# B&R Automation Studio project Parker_BMM_ST_V5_3147_V12 (part 21)

```c
					/*-------------F5---------*/
					//					gPanelObj.idxKeyPicture[S$KEYMATRIX_F5] = STATE_INACTIVE;
					gPanelObj.idxKeyPicture[S$KEYMATRIX_F5] = STATE_SUB_PAGE;
					if(1 == EDGEPOS(gPanelObj.KeyMatric[S$KEYMATRIX_F5],KeyMatric[S$KEYMATRIX_F5]))
					{
					gPanelObj.SetPicture = PIC_BLOW_PIN_CONFIG;
				}
				if(gPanelObj.GetPicture == PIC_BLOW_PIN_CONFIG)gPanelObj.idxKeyPicture[S$KEYMATRIX_F5] = STATE_ACTIVE;

					/*------------F6-----------*/
					gPanelObj.idxKeyPicture[S$KEYMATRIX_F6] = STATE_SUB_PAGE;
					if(1 == EDGEPOS(gPanelObj.KeyMatric[S$KEYMATRIX_F6],KeyMatric[S$KEYMATRIX_F6]))
					{
					gPanelObj.SetPicture = PIC_EXTRLIFT_CONFIG;
				}
				if(gPanelObj.GetPicture == PIC_EXTRLIFT_CONFIG)gPanelObj.idxKeyPicture[S$KEYMATRIX_F6] = STATE_ACTIVE;

					/*------------F7-----------*/
					gPanelObj.idxKeyPicture[S$KEYMATRIX_F7] = STATE_INACTIVE;

					/*-----------F8------------*/
					gPanelObj.idxKeyPicture[S$KEYMATRIX_F8] = STATE_INACTIVE;

					/*----------F9-------------*/
					gPanelObj.idxKeyPicture[S$KEYMATRIX_F9] = STATE_INACTIVE;

					/*----------F10-------------*/
					gPanelObj.idxKeyPicture[S$KEYMATRIX_F10] = STATE_INACTIVE;

					/*----------F11-------------*/
					gPanelObj.idxKeyPicture[S$KEYMATRIX_F11] = STATE_SUB_PAGE;
					if(1 == EDGEPOS(gPanelObj.KeyMatric[S$KEYMATRIX_F11],KeyMatric[S$KEYMATRIX_F11]))
					{
					gPanelObj.SetPicture = PIC_CLAMP_TOGGLE;
				}
				if(gPanelObj.GetPicture == PIC_CLAMP_TOGGLE)gPanelObj.idxKeyPicture[S$KEYMATRIX_F11] = STATE_ACTIVE;

					/*----------F12-------------*/
					gPanelObj.idxKeyPicture[S$KEYMATRIX_F12] = STATE_SUB_PAGE;
					if(1 == EDGEPOS(gPanelObj.KeyMatric[S$KEYMATRIX_F12],KeyMatric[S$KEYMATRIX_F12]))
					{
					gPanelObj.SetPicture = PIC_CARRIAGE_TOGGLE;
				}
				if(gPanelObj.GetPicture == PIC_CARRIAGE_TOGGLE)gPanelObj.idxKeyPicture[S$KEYMATRIX_F12] = STATE_ACTIVE;

					/*----------F13-------------*/
					gPanelObj.idxKeyPicture[S$KEYMATRIX_F13] = STATE_SUB_PAGE;
					if(1 == EDGEPOS(gPanelObj.KeyMatric[S$KEYMATRIX_F13],KeyMatric[S$KEYMATRIX_F13]))
					{
					gPanelObj.SetPicture = PIC_EXTRLIFT_TOGGLE;
				}
				if(gPanelObj.GetPicture == PIC_EXTRLIFT_TOGGLE)gPanelObj.idxKeyPicture[S$KEYMATRIX_F13] = STATE_ACTIVE;

					/*----------F14-------------*/
					gPanelObj.idxKeyPicture[S$KEYMATRIX_F14] = STATE_SUB_PAGE;
					if(1 == EDGEPOS(gPanelObj.KeyMatric[S$KEYMATRIX_F14],KeyMatric[S$KEYMATRIX_F14]))
					{
					gPanelObj.SetPicture = PIC_CONFIG_HELP;
				}
				if(gPanelObj.GetPicture == PIC_CONFIG_HELP)gPanelObj.idxKeyPicture[S$KEYMATRIX_F14] = STATE_ACTIVE;

					/*----------F15-------------*/
					gPanelObj.idxKeyPicture[S$KEYMATRIX_F15] = STATE_SUB_PAGE;
					if(1 == EDGEPOS(gPanelObj.KeyMatric[S$KEYMATRIX_F15],KeyMatric[S$KEYMATRIX_F15]))
					{
					gPanelObj.SetPicture = PIC_CLAMP_L;
					if(1 == bHideLeftStation)gPanelObj.SetPicture = PIC_CLAMP_R;
				}

				/*----------F16-------------*/
				gPanelObj.idxKeyPicture[S$KEYMATRIX_F16] = STATE_SUB_PAGE;
					if(1 == EDGEPOS(gPanelObj.KeyMatric[S$KEYMATRIX_F16],KeyMatric[S$KEYMATRIX_F16]))
					{
					gPanelObj.SetPicture = PIC_PASSWORD_LOGIN;
				}

				break;

			case PIC_RECIPE:
				if(ChangePageDly > 0)
				{
					ChangePageDly--;
					break;
				}

				gPanelObj.idxKeyPicture[S$KEYMATRIX_F1] = STATE_SUB_PAGE;
					if(1 == EDGEPOS(gPanelObj.KeyMatric[S$KEYMATRIX_F1],KeyMatric[S$KEYMATRIX_F1]))
					{
					gPanelObj.SetPicture = PIC_OVERVIEW;
				}

				gPanelObj.idxKeyPicture[S$KEYMATRIX_F2] = STATE_SUB_PAGE;
					if(1 == EDGEPOS(gPanelObj.KeyMatric[S$KEYMATRIX_F2],KeyMatric[S$KEYMATRIX_F2]))
					{
					gPanelObj.SetPicture = gPanelObj.OldPicture;
				}

				gPanelObj.idxKeyPicture[S$KEYMATRIX_F3] = STATE_INACTIVE;

					if(1 == gRecipeOperate.usbDiskOk)
				{
					gPanelObj.idxKeyPicture[S$KEYMATRIX_F4] = STATE_SUB_BUTTON;
						gPanelObj.idxKeyPicture[S$KEYMATRIX_F5] = STATE_SUB_BUTTON;
						}
				else
				{
					gPanelObj.idxKeyPicture[S$KEYMATRIX_F4] = STATE_INACTIVE;
						gPanelObj.idxKeyPicture[S$KEYMATRIX_F5] = STATE_INACTIVE;
						}
				gPanelObj.idxKeyPicture[S$KEYMATRIX_F6] = STATE_INACTIVE;

					gPanelObj.idxKeyPicture[S$KEYMATRIX_F7] = STATE_INACTIVE;
					gPanelObj.idxKeyPicture[S$KEYMATRIX_F8] = STATE_INACTIVE;
					gPanelObj.idxKeyPicture[S$KEYMATRIX_F9] = STATE_INACTIVE;
					gPanelObj.idxKeyPicture[S$KEYMATRIX_F10] = STATE_INACTIVE;
					gPanelObj.idxKeyPicture[S$KEYMATRIX_F11] = STATE_SUB_BUTTON;
					gPanelObj.idxKeyPicture[S$KEYMATRIX_F12] = STATE_SUB_BUTTON;
					gPanelObj.idxKeyPicture[S$KEYMATRIX_F13] = STATE_SUB_BUTTON;
					gPanelObj.idxKeyPicture[S$KEYMATRIX_F14] = STATE_SUB_BUTTON;

					gPanelObj.idxKeyPicture[S$KEYMATRIX_F15] = STATE_INACTIVE;

					gPanelObj.idxKeyPicture[S$KEYMATRIX_F16] = STATE_SUB_PAGE;
					if(1 == EDGEPOS(gPanelObj.KeyMatric[S$KEYMATRIX_F16],KeyMatric[S$KEYMATRIX_F16]))
					{
					gPanelObj.SetPicture = PIC_PASSWORD_LOGIN;
				}
				break;

			//				case PIC_SPEED:
			//					if(ChangePageDly > 0)
			//					{
			//						ChangePageDly--;
			//						break;
			//					}
			//
			//					gPanelObj.idxKeyPicture[S$KEYMATRIX_F1] = STATE_SUB_PAGE;
			//						if(1 == EDGEPOS(gPanelObj.KeyMatric[S$KEYMATRIX_F1],KeyMatric[S$KEYMATRIX_F1]))
			//						{
			//						gPanelObj.SetPicture = PIC_OVERVIEW;
			//					}
			//
			//					gPanelObj.idxKeyPicture[S$KEYMATRIX_F2] = STATE_SUB_PAGE;
			//						if(1 == EDGEPOS(gPanelObj.KeyMatric[S$KEYMATRIX_F2],KeyMatric[S$KEYMATRIX_F2]))
			//						{
			//						gPanelObj.SetPicture = gPanelObj.OldPicture;
			//					}
			//
			//					gPanelObj.idxKeyPicture[S$KEYMATRIX_F3] = STATE_INACTIVE;
			////						if(1 == EDGEPOS(gPanelObj.KeyMatric[S$KEYMATRIX_F3],KeyMatric[S$KEYMATRIX_F3]))
			////						{
			////						gPanelObj.SetPicture =PIC_LENGTH;
			////					}
			//
			//					gPanelObj.idxKeyPicture[S$KEYMATRIX_F4] = STATE_INACTIVE;
			//						gPanelObj.idxKeyPicture[S$KEYMATRIX_F5] = STATE_INACTIVE;
			//						gPanelObj.idxKeyPicture[S$KEYMATRIX_F6] = STATE_INACTIVE;
			//						gPanelObj.idxKeyPicture[S$KEYMATRIX_F7] = STATE_INACTIVE;
			//						gPanelObj.idxKeyPicture[S$KEYMATRIX_F8] = STATE_INACTIVE;
			//
			//						gPanelObj.idxKeyPicture[S$KEYMATRIX_F9] = STATE_SUB_PAGE;
			//						if(1 == EDGEPOS(gPanelObj.KeyMatric[S$KEYMATRIX_F9],KeyMatric[S$KEYMATRIX_F9]))
			//						{
			//						gPanelObj.SetPicture = PIC_TEMP_CONSTRUCT;
			//					}
			//
			//					gPanelObj.idxKeyPicture[S$KEYMATRIX_F10] = STATE_SUB_PAGE;
			//						if(1 == EDGEPOS(gPanelObj.KeyMatric[S$KEYMATRIX_F10],KeyMatric[S$KEYMATRIX_F10]))
			//						{
			//						gPanelObj.SetPicture =PIC_THICK_START;
			//					}
			//
			//					gPanelObj.idxKeyPicture[S$KEYMATRIX_F11] = STATE_INACTIVE;
			//						gPanelObj.idxKeyPicture[S$KEYMATRIX_F12] = STATE_INACTIVE;
			//						gPanelObj.idxKeyPicture[S$KEYMATRIX_F13] = STATE_INACTIVE;
			//						gPanelObj.idxKeyPicture[S$KEYMATRIX_F14] = STATE_INACTIVE;
			//						gPanelObj.idxKeyPicture[S$KEYMATRIX_F15] = STATE_INACTIVE;
			//
			//						gPanelObj.idxKeyPicture[S$KEYMATRIX_F16] = STATE_SUB_PAGE;
			//						if(1 == EDGEPOS(gPanelObj.KeyMatric[S$KEYMATRIX_F16],KeyMatric[S$KEYMATRIX_F16]))
			//						{
			//						gPanelObj.SetPicture = PIC_PASSWORD_LOGIN;
			//					}
			//					break;

			case PIC_LENGTH:
				if(ChangePageDly > 0)
				{
					ChangePageDly--;
					break;
				}

				gPanelObj.idxKeyPicture[S$KEYMATRIX_F1] = STATE_SUB_PAGE;
					if(1 == EDGEPOS(gPanelObj.KeyMatric[S$KEYMATRIX_F1],KeyMatric[S$KEYMATRIX_F1]))
					{
					gPanelObj.SetPicture = PIC_OVERVIEW;
				}

				gPanelObj.idxKeyPicture[S$KEYMATRIX_F2] = STATE_SUB_PAGE;
					if(1 == EDGEPOS(gPanelObj.KeyMatric[S$KEYMATRIX_F2],KeyMatric[S$KEYMATRIX_F2]))
					{
					gPanelObj.SetPicture =PIC_SPEED;
				}

				gPanelObj.idxKeyPicture[S$KEYMATRIX_F3] = STATE_SUB_PAGE;
					if(1 == EDGEPOS(gPanelObj.KeyMatric[S$KEYMATRIX_F3],KeyMatric[S$KEYMATRIX_F3]))
					{
					gPanelObj.SetPicture =PIC_SPEED;
				}

				gPanelObj.idxKeyPicture[S$KEYMATRIX_F4] = STATE_INACTIVE;
					gPanelObj.idxKeyPicture[S$KEYMATRIX_F5] = STATE_INACTIVE;
					gPanelObj.idxKeyPicture[S$KEYMATRIX_F6] = STATE_INACTIVE;
					gPanelObj.idxKeyPicture[S$KEYMATRIX_F7] = STATE_INACTIVE;
					gPanelObj.idxKeyPicture[S$KEYMATRIX_F8] = STATE_INACTIVE;
					gPanelObj.idxKeyPicture[S$KEYMATRIX_F9] = STATE_INACTIVE;

					gPanelObj.idxKeyPicture[S$KEYMATRIX_F10] = STATE_SUB_BUTTON;
					if(1 == EDGEPOS(gPanelObj.KeyMatric[S$KEYMATRIX_F10],KeyMatric[S$KEYMATRIX_F10]))
					{
					gMachinePara.LengthPara.LengthEnable = !gMachinePara.LengthPara.LengthEnable;
				}

				gPanelObj.idxKeyPicture[S$KEYMATRIX_F11] = STATE_INACTIVE;
					gPanelObj.idxKeyPicture[S$KEYMATRIX_F12] = STATE_INACTIVE;
					gPanelObj.idxKeyPicture[S$KEYMATRIX_F13] = STATE_INACTIVE;
					gPanelObj.idxKeyPicture[S$KEYMATRIX_F14] = STATE_INACTIVE;
					gPanelObj.idxKeyPicture[S$KEYMATRIX_F15] = STATE_INACTIVE;

					gPanelObj.idxKeyPicture[S$KEYMATRIX_F16] = STATE_SUB_PAGE;
					if(1 == EDGEPOS(gPanelObj.KeyMatric[S$KEYMATRIX_F16],KeyMatric[S$KEYMATRIX_F16]))
					{
					gPanelObj.SetPicture = PIC_PASSWORD_LOGIN;
				}
				break;

			case PIC_THICK_START:
			case PIC_THICK_DIVER:

				if(1 == gThickProf.FunOption.SealMode) bHideSealGap = 0;
				else bHideSealGap = 1;

				if(ChangePageDly > 0)
				{
				ChangePageDly--;
				break;
				}

				gPanelObj.idxKeyPicture[S$KEYMATRIX_F1] = STATE_SUB_PAGE;
					if(1 == EDGEPOS(gPanelObj.KeyMatric[S$KEYMATRIX_F1],KeyMatric[S$KEYMATRIX_F1]))
					{
					gPanelObj.SetPicture = PIC_OVERVIEW;
				}

				gPanelObj.idxKeyPicture[S$KEYMATRIX_F2] = STATE_SUB_PAGE;
					if(1 == EDGEPOS(gPanelObj.KeyMatric[S$KEYMATRIX_F2],KeyMatric[S$KEYMATRIX_F2]))
					{
					gPanelObj.SetPicture = gPanelObj.OldPicture;
				}

				gPanelObj.idxKeyPicture[S$KEYMATRIX_F3] = STATE_ACTIVE;
					if(1 == EDGEPOS(gPanelObj.KeyMatric[S$KEYMATRIX_F3],KeyMatric[S$KEYMATRIX_F3]))
					{
					gPanelObj.SetPicture = PIC_THICK_START;
				}

				gPanelObj.idxKeyPicture[S$KEYMATRIX_F4] = STATE_SUB_PAGE;
					if(1 == EDGEPOS(gPanelObj.KeyMatric[S$KEYMATRIX_F4],KeyMatric[S$KEYMATRIX_F4]))
					{
					gPanelObj.SetPicture = PIC_CURVE_EDIT;
				}

				gPanelObj.idxKeyPicture[S$KEYMATRIX_F5] = STATE_SUB_PAGE;
					if(1 == EDGEPOS(gPanelObj.KeyMatric[S$KEYMATRIX_F5],KeyMatric[S$KEYMATRIX_F5]))
					{
					gPanelObj.SetPicture = PIC_CURVE_TRACE;
				}

				gPanelObj.idxKeyPicture[S$KEYMATRIX_F6] = STATE_SUB_PAGE;
					if(1 == EDGEPOS(gPanelObj.KeyMatric[S$KEYMATRIX_F6],KeyMatric[S$KEYMATRIX_F6]))
					{
					gPanelObj.SetPicture = PIC_MARKER_SET_A;
				}

				gPanelObj.idxKeyPicture[S$KEYMATRIX_F7] = STATE_SUB_PAGE;
					if(1 == EDGEPOS(gPanelObj.KeyMatric[S$KEYMATRIX_F7],KeyMatric[S$KEYMATRIX_F7]))
					{
					gPanelObj.SetPicture = PIC_CURVEDATA_A;
				}

				gPanelObj.idxKeyPicture[S$KEYMATRIX_F8] = STATE_SUB_PAGE;
					if(1 == EDGEPOS(gPanelObj.KeyMatric[S$KEYMATRIX_F8],KeyMatric[S$KEYMATRIX_F8]))
					{
					gPanelObj.SetPicture = PIC_TEMP_CONSTRUCT;
				}

				gPanelObj.idxKeyPicture[S$KEYMATRIX_F9] = STATE_SUB_PAGE;
					if(1 == EDGEPOS(gPanelObj.KeyMatric[S$KEYMATRIX_F9],KeyMatric[S$KEYMATRIX_F9]))
					{
					gPanelObj.SetPicture = PIC_SPEED;
				}
				gPanelObj.idxKeyPicture[S$KEYMATRIX_F10] = STATE_INACTIVE;
					gPanelObj.idxKeyPicture[S$KEYMATRIX_F11] = STATE_INACTIVE;
					gPanelObj.idxKeyPicture[S$KEYMATRIX_F12] = STATE_SUB_PAGE;
					if(1 == EDGEPOS(gPanelObj.KeyMatric[S$KEYMATRIX_F12],KeyMatric[S$KEYMATRIX_F12]))
					{
					gPanelObj.SetPicture = PIC_THICK_DIVER;
				}
				gPanelObj.idxKeyPicture[S$KEYMATRIX_F13] = STATE_SUB_PAGE;
					if(1 == EDGENEG(gPanelObj.KeyMatric[S$KEYMATRIX_F13],KeyMatric[S$KEYMATRIX_F13]))
					{
					//	if(gPanelObj.PasswordLevel > 2 &&  1 == gTKcalib.Status)
					if(gPanelObj.PasswordLevel > 2 &&  0 == gTKauto.Status)

					{
						gPanelObj.SetPicture = PIC_INIT_SET  ;
						OldSet    = gThickProf.ShareSet;
						OldFunSet = gThickProf.FunOption;
					}
				}
				//	if(1 == bThickCalibHide)gPanelObj.idxKeyPicture[S$KEYMATRIX_F13] = STATE_INACTIVE;
				if(1 == gTKauto.Status)gPanelObj.idxKeyPicture[S$KEYMATRIX_F13] = STATE_INACTIVE;

					gPanelObj.idxKeyPicture[S$KEYMATRIX_F14] = STATE_SUB_PAGE;
					if(1 == EDGENEG(gPanelObj.KeyMatric[S$KEYMATRIX_F14],KeyMatric[S$KEYMATRIX_F14]))
					{
					//	if(gPanelObj.PasswordLevel > 2 &&  1 == gTKcalib.Status)
					if(gPanelObj.PasswordLevel > 2 &&  0 == gTKauto.Status)
					{
						gPanelObj.SetPicture = PIC_GAP_CALIBRATE;
						OldSet    = gThickProf.ShareSet;
						OldFunSet = gThickProf.FunOption;
					}
				}
				//if(1 == bThickCalibHide)gPanelObj.idxKeyPicture[S$KEYMATRIX_F14] = STATE_INACTIVE;
				if(1 == gTKauto.Status)gPanelObj.idxKeyPicture[S$KEYMATRIX_F14] = STATE_INACTIVE;
					gPanelObj.idxKeyPicture[S$KEYMATRIX_F15] = STATE_SUB_BUTTON;
					gPanelObj.idxKeyPicture[S$KEYMATRIX_F16] = STATE_SUB_PAGE;
					if(1 == EDGEPOS(gPanelObj.KeyMatric[S$KEYMATRIX_F16],KeyMatric[S$KEYMATRIX_F16]))
					{
					gPanelObj.SetPicture = PIC_PASSWORD_LOGIN;
				}
				break;

			case PIC_CURVE_TRACE:
				if(ChangePageDly > 0)
				{
					ChangePageDly--;
					break;
				}

				gPanelObj.idxKeyPicture[S$KEYMATRIX_F1] = STATE_SUB_PAGE;
					if(1 == EDGEPOS(gPanelObj.KeyMatric[S$KEYMATRIX_F1],KeyMatric[S$KEYMATRIX_F1]))
					{
					gPanelObj.SetPicture = PIC_OVERVIEW;
				}

				gPanelObj.idxKeyPicture[S$KEYMATRIX_F2] = STATE_SUB_PAGE;
					if(1 == EDGEPOS(gPanelObj.KeyMatric[S$KEYMATRIX_F2],KeyMatric[S$KEYMATRIX_F2]))
					{
					gPanelObj.SetPicture = gPanelObj.OldPicture;
				}

				gPanelObj.idxKeyPicture[S$KEYMATRIX_F3] = STATE_ACTIVE;
					if(1 == EDGEPOS(gPanelObj.KeyMatric[S$KEYMATRIX_F3],KeyMatric[S$KEYMATRIX_F3]))
					{
					gPanelObj.SetPicture = PIC_THICK_START;
				}

				gPanelObj.idxKeyPicture[S$KEYMATRIX_F4] = STATE_SUB_PAGE;
					if(1 == EDGEPOS(gPanelObj.KeyMatric[S$KEYMATRIX_F4],KeyMatric[S$KEYMATRIX_F4]))
					{
					gPanelObj.SetPicture = PIC_CURVE_EDIT;
				}

				gPanelObj.idxKeyPicture[S$KEYMATRIX_F5] = STATE_SUB_PAGE;
					if(1 == EDGEPOS(gPanelObj.KeyMatric[S$KEYMATRIX_F5],KeyMatric[S$KEYMATRIX_F5]))
					{
					gPanelObj.SetPicture = PIC_CURVE_TRACE;
				}

				gPanelObj.idxKeyPicture[S$KEYMATRIX_F6] = STATE_SUB_PAGE;
					if(1 == EDGEPOS(gPanelObj.KeyMatric[S$KEYMATRIX_F6],KeyMatric[S$KEYMATRIX_F6]))
					{
					gPanelObj.SetPicture = PIC_MARKER_SET_A;
				}

				gPanelObj.idxKeyPicture[S$KEYMATRIX_F7] = STATE_SUB_PAGE;
					if(1 == EDGEPOS(gPanelObj.KeyMatric[S$KEYMATRIX_F7],KeyMatric[S$KEYMATRIX_F7]))
					{
					gPanelObj.SetPicture = PIC_CURVEDATA_A;
				}

				gPanelObj.idxKeyPicture[S$KEYMATRIX_F8] = STATE_SUB_PAGE;
					if(1 == EDGEPOS(gPanelObj.KeyMatric[S$KEYMATRIX_F8],KeyMatric[S$KEYMATRIX_F8]))
					{
					gPanelObj.SetPicture = PIC_TEMP_CONSTRUCT;
				}

				gPanelObj.idxKeyPicture[S$KEYMATRIX_F9] = STATE_SUB_PAGE;
					if(1 == EDGEPOS(gPanelObj.KeyMatric[S$KEYMATRIX_F9],KeyMatric[S$KEYMATRIX_F9]))
					{
					gPanelObj.SetPicture = PIC_SPEED;
				}

				gPanelObj.idxKeyPicture[S$KEYMATRIX_F10] = STATE_INACTIVE;
					gPanelObj.idxKeyPicture[S$KEYMATRIX_F11] = STATE_INACTIVE;
					if(1 == EDGEPOS(gPanelObj.KeyMatric[S$KEYMATRIX_F12],KeyMatric[S$KEYMATRIX_F12]))
					{
					gPanelObj.SetPicture = PIC_THICK_DIVER;
				}
				gPanelObj.idxKeyPicture[S$KEYMATRIX_F13] = STATE_SUB_PAGE;
					if(1 == EDGENEG(gPanelObj.KeyMatric[S$KEYMATRIX_F13],KeyMatric[S$KEYMATRIX_F13]))
					{
					//	if(gPanelObj.PasswordLevel > 2 &&  1 == gTKcalib.Status)
					if(gPanelObj.PasswordLevel > 2 &&  0 == gTKauto.Status)
					{
						gPanelObj.SetPicture = PIC_INIT_SET  ;
						OldSet    = gThickProf.ShareSet;
						OldFunSet = gThickProf.FunOption;
					}
				}
				//	if(1 == bThickCalibHide)gPanelObj.idxKeyPicture[S$KEYMATRIX_F13] = STATE_INACTIVE;
				if(1 == gTKauto.Status)gPanelObj.idxKeyPicture[S$KEYMATRIX_F13] = STATE_INACTIVE;

					gPanelObj.idxKeyPicture[S$KEYMATRIX_F14] = STATE_SUB_PAGE;
					if(1 == EDGENEG(gPanelObj.KeyMatric[S$KEYMATRIX_F14],KeyMatric[S$KEYMATRIX_F14]))
					{
					//	if(gPanelObj.PasswordLevel > 2 &&  1 == gTKcalib.Status)
					if(gPanelObj.PasswordLevel > 2 &&  0 == gTKauto.Status)
					{
						gPanelObj.SetPicture = PIC_GAP_CALIBRATE;
						OldSet    = gThickProf.ShareSet;
						OldFunSet = gThickProf.FunOption;
					}
				}
				//if(1 == bThickCalibHide)gPanelObj.idxKeyPicture[S$KEYMATRIX_F14] = STATE_INACTIVE;
				if(1 == gTKauto.Status)gPanelObj.idxKeyPicture[S$KEYMATRIX_F14] = STATE_INACTIVE;
					//						gPanelObj.idxKeyPicture[S$KEYMATRIX_F13] = STATE_INACTIVE;
					//						gPanelObj.idxKeyPicture[S$KEYMATRIX_F14] = STATE_INACTIVE;
					gPanelObj.idxKeyPicture[S$KEYMATRIX_F15] = STATE_INACTIVE;
					gPanelObj.idxKeyPicture[S$KEYMATRIX_F16] = STATE_SUB_PAGE;
					if(1 == EDGEPOS(gPanelObj.KeyMatric[S$KEYMATRIX_F16],KeyMatric[S$KEYMATRIX_F16]))
					{
					gPanelObj.SetPicture = PIC_PASSWORD_LOGIN;
				}
				break;

			case PIC_CURVE_EDIT:
				if(ChangePageDly > 0)
				{
					ChangePageDly--;
					break;
				}

				gPanelObj.idxKeyPicture[S$KEYMATRIX_F1] = STATE_SUB_PAGE;
					if(1 == EDGEPOS(gPanelObj.KeyMatric[S$KEYMATRIX_F1],KeyMatric[S$KEYMATRIX_F1]))
					{
					gPanelObj.SetPicture = PIC_OVERVIEW;
				}

				gPanelObj.idxKeyPicture[S$KEYMATRIX_F2] = STATE_SUB_PAGE;
					if(1 == EDGEPOS(gPanelObj.KeyMatric[S$KEYMATRIX_F2],KeyMatric[S$KEYMATRIX_F2]))
					{
					gPanelObj.SetPicture = gPanelObj.OldPicture;
				}

				gPanelObj.idxKeyPicture[S$KEYMATRIX_F3] = STATE_ACTIVE;
					if(1 == EDGEPOS(gPanelObj.KeyMatric[S$KEYMATRIX_F3],KeyMatric[S$KEYMATRIX_F3]))
					{
					gPanelObj.SetPicture = PIC_THICK_START;
				}

				gPanelObj.idxKeyPicture[S$KEYMATRIX_F4] = STATE_SUB_PAGE;
					if(1 == EDGEPOS(gPanelObj.KeyMatric[S$KEYMATRIX_F4],KeyMatric[S$KEYMATRIX_F4]))
					{
					gPanelObj.SetPicture = PIC_CURVE_EDIT;
				}

				gPanelObj.idxKeyPicture[S$KEYMATRIX_F5] = STATE_SUB_PAGE;
					if(1 == EDGEPOS(gPanelObj.KeyMatric[S$KEYMATRIX_F5],KeyMatric[S$KEYMATRIX_F5]))
					{
					gPanelObj.SetPicture = PIC_CURVE_TRACE;
				}

				gPanelObj.idxKeyPicture[S$KEYMATRIX_F6] = STATE_SUB_PAGE;
					if(1 == EDGEPOS(gPanelObj.KeyMatric[S$KEYMATRIX_F6],KeyMatric[S$KEYMATRIX_F6]))
					{
					gPanelObj.SetPicture = PIC_MARKER_SET_A;
				}

				gPanelObj.idxKeyPicture[S$KEYMATRIX_F7] = STATE_SUB_PAGE;
					if(1 == EDGEPOS(gPanelObj.KeyMatric[S$KEYMATRIX_F7],KeyMatric[S$KEYMATRIX_F7]))
					{
					gPanelObj.SetPicture = PIC_CURVEDATA_A;
				}

				gPanelObj.idxKeyPicture[S$KEYMATRIX_F8] = STATE_SUB_PAGE;
					if(1 == EDGEPOS(gPanelObj.KeyMatric[S$KEYMATRIX_F8],KeyMatric[S$KEYMATRIX_F8]))
					{
					gPanelObj.SetPicture = PIC_TEMP_CONSTRUCT;
				}

				gPanelObj.idxKeyPicture[S$KEYMATRIX_F9] = STATE_SUB_PAGE;
					if(1 == EDGEPOS(gPanelObj.KeyMatric[S$KEYMATRIX_F9],KeyMatric[S$KEYMATRIX_F9]))
					{
					gPanelObj.SetPicture = PIC_SPEED;
				}
				gPanelObj.idxKeyPicture[S$KEYMATRIX_F10] = STATE_INACTIVE;
					gPanelObj.idxKeyPicture[S$KEYMATRIX_F11] = STATE_INACTIVE;
					if(1 == EDGEPOS(gPanelObj.KeyMatric[S$KEYMATRIX_F12],KeyMatric[S$KEYMATRIX_F12]))
					{
					gPanelObj.SetPicture = PIC_THICK_DIVER;
				}
				gPanelObj.idxKeyPicture[S$KEYMATRIX_F13] = STATE_SUB_PAGE;
					if(1 == EDGENEG(gPanelObj.KeyMatric[S$KEYMATRIX_F13],KeyMatric[S$KEYMATRIX_F13]))
					{
					//	if(gPanelObj.PasswordLevel > 2 &&  1 == gTKcalib.Status)
					if(gPanelObj.PasswordLevel > 2 &&  0 == gTKauto.Status)
					{
						gPanelObj.SetPicture = PIC_INIT_SET  ;
						OldSet    = gThickProf.ShareSet;
						OldFunSet = gThickProf.FunOption;
					}
				}
				if(1 == gTKauto.Status)gPanelObj.idxKeyPicture[S$KEYMATRIX_F13] = STATE_INACTIVE;

					gPanelObj.idxKeyPicture[S$KEYMATRIX_F14] = STATE_SUB_PAGE;
					if(1 == EDGENEG(gPanelObj.KeyMatric[S$KEYMATRIX_F14],KeyMatric[S$KEYMATRIX_F14]))
					{
					//	if(gPanelObj.PasswordLevel > 2 &&  1 == gTKcalib.Status)
					if(gPanelObj.PasswordLevel > 2 &&  0 == gTKauto.Status)
					{
						gPanelObj.SetPicture = PIC_GAP_CALIBRATE;
						OldSet    = gThickProf.ShareSet;
						OldFunSet = gThickProf.FunOption;
					}
				}
				if(1 == gTKauto.Status)gPanelObj.idxKeyPicture[S$KEYMATRIX_F14] = STATE_INACTIVE;
					//						gPanelObj.idxKeyPicture[S$KEYMATRIX_F13] = STATE_INACTIVE;
					//						gPanelObj.idxKeyPicture[S$KEYMATRIX_F14] = STATE_INACTIVE;
					gPanelObj.idxKeyPicture[S$KEYMATRIX_F15] = STATE_SUB_BUTTON;
					if(1 == EDGEPOS(gPanelObj.KeyMatric[S$KEYMATRIX_F16],KeyMatric[S$KEYMATRIX_F16]))
					{
					gPanelObj.SetPicture = PIC_PASSWORD_LOGIN;
				}
				break;

			case PIC_MARKER_SET_A:
				if(ChangePageDly > 0)
				{
					ChangePageDly--;
					break;
				}

				gPanelObj.idxKeyPicture[S$KEYMATRIX_F1] = STATE_SUB_PAGE;
					if(1 == EDGEPOS(gPanelObj.KeyMatric[S$KEYMATRIX_F1],KeyMatric[S$KEYMATRIX_F1]))
					{
					gPanelObj.SetPicture = PIC_OVERVIEW;
				}

				gPanelObj.idxKeyPicture[S$KEYMATRIX_F2] = STATE_SUB_PAGE;
					if(1 == EDGEPOS(gPanelObj.KeyMatric[S$KEYMATRIX_F2],KeyMatric[S$KEYMATRIX_F2]))
					{
					gPanelObj.SetPicture = gPanelObj.OldPicture;
				}

				gPanelObj.idxKeyPicture[S$KEYMATRIX_F3] = STATE_ACTIVE;
					if(1 == EDGEPOS(gPanelObj.KeyMatric[S$KEYMATRIX_F3],KeyMatric[S$KEYMATRIX_F3]))
					{
					gPanelObj.SetPicture = PIC_THICK_START;
				}

				gPanelObj.idxKeyPicture[S$KEYMATRIX_F4] = STATE_SUB_PAGE;
					if(1 == EDGEPOS(gPanelObj.KeyMatric[S$KEYMATRIX_F4],KeyMatric[S$KEYMATRIX_F4]))
					{
					gPanelObj.SetPicture = PIC_CURVE_EDIT;
				}

				gPanelObj.idxKeyPicture[S$KEYMATRIX_F5] = STATE_SUB_PAGE;
					if(1 == EDGEPOS(gPanelObj.KeyMatric[S$KEYMATRIX_F5],KeyMatric[S$KEYMATRIX_F5]))
					{
					gPanelObj.SetPicture = PIC_CURVE_TRACE;
				}

				gPanelObj.idxKeyPicture[S$KEYMATRIX_F6] = STATE_SUB_PAGE;
					if(1 == EDGEPOS(gPanelObj.KeyMatric[S$KEYMATRIX_F6],KeyMatric[S$KEYMATRIX_F6]))
					{
					gPanelObj.SetPicture = PIC_MARKER_SET_A;
				}

				gPanelObj.idxKeyPicture[S$KEYMATRIX_F7] = STATE_SUB_PAGE;
					if(1 == EDGEPOS(gPanelObj.KeyMatric[S$KEYMATRIX_F7],KeyMatric[S$KEYMATRIX_F7]))
					{
					gPanelObj.SetPicture = PIC_CURVEDATA_A;
				}

				gPanelObj.idxKeyPicture[S$KEYMATRIX_F8] = STATE_SUB_PAGE;
					if(1 == EDGEPOS(gPanelObj.KeyMatric[S$KEYMATRIX_F8],KeyMatric[S$KEYMATRIX_F8]))
					{
					gPanelObj.SetPicture = PIC_TEMP_CONSTRUCT;
				}

				gPanelObj.idxKeyPicture[S$KEYMATRIX_F9] = STATE_SUB_PAGE;
					if(1 == EDGEPOS(gPanelObj.KeyMatric[S$KEYMATRIX_F9],KeyMatric[S$KEYMATRIX_F9]))
					{
					gPanelObj.SetPicture = PIC_SPEED;
				}
				gPanelObj.idxKeyPicture[S$KEYMATRIX_F10] = STATE_INACTIVE;
					gPanelObj.idxKeyPicture[S$KEYMATRIX_F11] = STATE_INACTIVE;
					if(1 == EDGEPOS(gPanelObj.KeyMatric[S$KEYMATRIX_F12],KeyMatric[S$KEYMATRIX_F12]))
					{
					gPanelObj.SetPicture = PIC_THICK_DIVER;
				}
				gPanelObj.idxKeyPicture[S$KEYMATRIX_F13] = STATE_SUB_PAGE;
					if(1 == EDGENEG(gPanelObj.KeyMatric[S$KEYMATRIX_F13],KeyMatric[S$KEYMATRIX_F13]))
					{
					//	if(gPanelObj.PasswordLevel > 2 &&  1 == gTKcalib.Status)
					if(gPanelObj.PasswordLevel > 2 &&  0 == gTKauto.Status)
					{
						gPanelObj.SetPicture = PIC_INIT_SET  ;
						OldSet    = gThickProf.ShareSet;
						OldFunSet = gThickProf.FunOption;
					}
				}
				if(1 == gTKauto.Status)gPanelObj.idxKeyPicture[S$KEYMATRIX_F13] = STATE_INACTIVE;

					gPanelObj.idxKeyPicture[S$KEYMATRIX_F14] = STATE_SUB_PAGE;
					if(1 == EDGENEG(gPanelObj.KeyMatric[S$KEYMATRIX_F14],KeyMatric[S$KEYMATRIX_F14]))
					{
					//	if(gPanelObj.PasswordLevel > 2 &&  1 == gTKcalib.Status)
					if(gPanelObj.PasswordLevel > 2 &&  0 == gTKauto.Status)
					{
						gPanelObj.SetPicture = PIC_GAP_CALIBRATE;
						OldSet    = gThickProf.ShareSet;
						OldFunSet = gThickProf.FunOption;
					}
				}
				if(1 == gTKauto.Status)gPanelObj.idxKeyPicture[S$KEYMATRIX_F14] = STATE_INACTIVE;
					//						gPanelObj.idxKeyPicture[S$KEYMATRIX_F13] = STATE_INACTIVE;
					//						gPanelObj.idxKeyPicture[S$KEYMATRIX_F14] = STATE_INACTIVE;
					gPanelObj.idxKeyPicture[S$KEYMATRIX_F15] = STATE_INACTIVE;

					gPanelObj.idxKeyPicture[S$KEYMATRIX_F16] = STATE_SUB_PAGE;
					if(1 == EDGEPOS(gPanelObj.KeyMatric[S$KEYMATRIX_F16],KeyMatric[S$KEYMATRIX_F16]))
					{
					gPanelObj.SetPicture = PIC_PASSWORD_LOGIN;
				}

				MarkerDis.Current = MarkerDis.Current % MarkerDis.Count;

				if(1 == EDGEPOS(gPanelObj.KeyMatric[S$KEYMATRIX_UP],KeyMatric[S$KEYMATRIX_UP])) /* UP ARROW  */
					{
					if(0 == MarkerDis.Current)
					{
						MarkerDis.Current = MarkerDis.Count - 1;
					}
					else
					{
						MarkerDis.Current--;
					}
				}

				if(1 == EDGEPOS(gPanelObj.KeyMatric[S$KEYMATRIX_DOWN],KeyMatric[S$KEYMATRIX_DOWN])) /* DOWN ARROW  */
					{
					if(MarkerDis.Current >= (MarkerDis.Count-1))
					{
						MarkerDis.Current = 0;
					}
					else
					{
						MarkerDis.Current++;
					}
				}

				if(1 == EDGEPOS(gPanelObj.KeyMatric[S$KEYMATRIX_LEFT],KeyMatric[S$KEYMATRIX_LEFT])) /* LEFT ARROW  */
					{
					MarkerDis.Current = MarkerDis.Current - MarkerDis.Section;
					if(MarkerDis.Current < 0)
					{
						MarkerDis.Current = MarkerDis.Current + MarkerDis.Count;
					}
				}

				if(1 == EDGEPOS(gPanelObj.KeyMatric[S$KEYMATRIX_RIGHT],KeyMatric[S$KEYMATRIX_RIGHT])) /* RIGHT ARROW  */
					{
					MarkerDis.Current = MarkerDis.Current + MarkerDis.Section;
					if(MarkerDis.Current > MarkerDis.Count - 1)
					{
						MarkerDis.Current = MarkerDis.Current - MarkerDis.Count;
					}
				}

				if(MarkerDis.Current >= MarkerDis.Count)MarkerDis.Current = 0;

				if(1 == EDGEPOS(gPanelObj.KeyMatric[S$KEYMATRIX_TAB],KeyMatric[S$KEYMATRIX_TAB]))
					{
					MarkerDis.pSource[MarkerDis.Current] = !MarkerDis.pSource[MarkerDis.Current];
				}

				for(i=0;i<100;i++)
				{
					MarkerDis.Obj[i] = MarkerDis.pSource[i];
				}

				MarkerDis.Obj[MarkerDis.Current] = MarkerDis.pSource[MarkerDis.Current] + 2;
				break;

			case PIC_CURVEDATA_A:
			case PIC_CURVEDATA_B:
				if(ChangePageDly > 0)
				{
					ChangePageDly--;
					break;
				}

				gPanelObj.idxKeyPicture[S$KEYMATRIX_F1] = STATE_SUB_PAGE;
					if(1 == EDGEPOS(gPanelObj.KeyMatric[S$KEYMATRIX_F1],KeyMatric[S$KEYMATRIX_F1]))
					{
					gPanelObj.SetPicture = PIC_OVERVIEW;
				}

				gPanelObj.idxKeyPicture[S$KEYMATRIX_F2] = STATE_SUB_PAGE;
					if(1 == EDGEPOS(gPanelObj.KeyMatric[S$KEYMATRIX_F2],KeyMatric[S$KEYMATRIX_F2]))
					{
					gPanelObj.SetPicture = gPanelObj.OldPicture;
				}

				gPanelObj.idxKeyPicture[S$KEYMATRIX_F3] = STATE_ACTIVE;
					if(1 == EDGEPOS(gPanelObj.KeyMatric[S$KEYMATRIX_F3],KeyMatric[S$KEYMATRIX_F3]))
					{
					gPanelObj.SetPicture = PIC_THICK_START;
				}

				gPanelObj.idxKeyPicture[S$KEYMATRIX_F4] = STATE_SUB_PAGE;
					if(1 == EDGEPOS(gPanelObj.KeyMatric[S$KEYMATRIX_F4],KeyMatric[S$KEYMATRIX_F4]))
					{
					gPanelObj.SetPicture = PIC_CURVE_EDIT;
				}

				gPanelObj.idxKeyPicture[S$KEYMATRIX_F5] = STATE_SUB_PAGE;
					if(1 == EDGEPOS(gPanelObj.KeyMatric[S$KEYMATRIX_F5],KeyMatric[S$KEYMATRIX_F5]))
					{
					gPanelObj.SetPicture = PIC_CURVE_TRACE;
				}

				gPanelObj.idxKeyPicture[S$KEYMATRIX_F6] = STATE_SUB_PAGE;
					if(1 == EDGEPOS(gPanelObj.KeyMatric[S$KEYMATRIX_F6],KeyMatric[S$KEYMATRIX_F6]))
					{
					gPanelObj.SetPicture = PIC_MARKER_SET_A;
				}

				gPanelObj.idxKeyPicture[S$KEYMATRIX_F7] = STATE_SUB_PAGE;
					if(1 == EDGEPOS(gPanelObj.KeyMatric[S$KEYMATRIX_F7],KeyMatric[S$KEYMATRIX_F7]))
					{
					gPanelObj.SetPicture = PIC_CURVEDATA_A;
				}

				gPanelObj.idxKeyPicture[S$KEYMATRIX_F8] = STATE_SUB_PAGE;
					if(1 == EDGEPOS(gPanelObj.KeyMatric[S$KEYMATRIX_F8],KeyMatric[S$KEYMATRIX_F8]))
					{
					gPanelObj.SetPicture = PIC_TEMP_CONSTRUCT;
				}

				gPanelObj.idxKeyPicture[S$KEYMATRIX_F9] = STATE_SUB_PAGE;
					if(1 == EDGEPOS(gPanelObj.KeyMatric[S$KEYMATRIX_F9],KeyMatric[S$KEYMATRIX_F9]))
					{
					gPanelObj.SetPicture = PIC_SPEED;
				}
				gPanelObj.idxKeyPicture[S$KEYMATRIX_F10] = STATE_INACTIVE;
					gPanelObj.idxKeyPicture[S$KEYMATRIX_F11] = STATE_INACTIVE;
					if(1 == EDGEPOS(gPanelObj.KeyMatric[S$KEYMATRIX_F12],KeyMatric[S$KEYMATRIX_F12]))
					{
					gPanelObj.SetPicture = PIC_THICK_DIVER;
				}
				gPanelObj.idxKeyPicture[S$KEYMATRIX_F13] = STATE_SUB_PAGE;
					if(1 == EDGENEG(gPanelObj.KeyMatric[S$KEYMATRIX_F13],KeyMatric[S$KEYMATRIX_F13]))
					{
					//	if(gPanelObj.PasswordLevel > 2 &&  1 == gTKcalib.Status)
					if(gPanelObj.PasswordLevel > 2 &&  0 == gTKauto.Status)
					{
						gPanelObj.SetPicture = PIC_INIT_SET  ;
						OldSet    = gThickProf.ShareSet;
						OldFunSet = gThickProf.FunOption;
					}
				}
				if(1 == gTKauto.Status)gPanelObj.idxKeyPicture[S$KEYMATRIX_F13] = STATE_INACTIVE;

					gPanelObj.idxKeyPicture[S$KEYMATRIX_F14] = STATE_SUB_PAGE;
					if(1 == EDGENEG(gPanelObj.KeyMatric[S$KEYMATRIX_F14],KeyMatric[S$KEYMATRIX_F14]))
					{
					//	if(gPanelObj.PasswordLevel > 2 &&  1 == gTKcalib.Status)
					if(gPanelObj.PasswordLevel > 2 &&  0 == gTKauto.Status)
					{
						gPanelObj.SetPicture = PIC_GAP_CALIBRATE;
						OldSet    = gThickProf.ShareSet;
						OldFunSet = gThickProf.FunOption;
					}
				}
				if(1 == gTKauto.Status)gPanelObj.idxKeyPicture[S$KEYMATRIX_F14] = STATE_INACTIVE;
					//						gPanelObj.idxKeyPicture[S$KEYMATRIX_F13] = STATE_INACTIVE;
					//						gPanelObj.idxKeyPicture[S$KEYMATRIX_F14] = STATE_INACTIVE;
					gPanelObj.idxKeyPicture[S$KEYMATRIX_F15] = STATE_INACTIVE;

					gPanelObj.idxKeyPicture[S$KEYMATRIX_F16] = STATE_SUB_PAGE;
					if(1 == EDGEPOS(gPanelObj.KeyMatric[S$KEYMATRIX_F16],KeyMatric[S$KEYMATRIX_F16]))
					{
					gPanelObj.SetPicture = PIC_PASSWORD_LOGIN;
				}
				break;

			case PIC_IO_DI_1:
			case PIC_IO_DI_2:
			case PIC_IO_DI_3:
			case PIC_IO_AI_1:
			case PIC_IO_MODULE:
			case PIC_IO_DRIVER_1:
			case PIC_IO_DRIVER_2:
			case PIC_ENERGY_MONITOR_ALL:
			case PIC_ENERGY_MONITOR:
			case PIC_MOTOR_TREND:
				if(ChangePageDly > 0)
				{
					ChangePageDly--;
					break;
				}

				gPanelObj.idxKeyPicture[S$KEYMATRIX_F1] = STATE_SUB_PAGE;
					if(1 == EDGEPOS(gPanelObj.KeyMatric[S$KEYMATRIX_F1],KeyMatric[S$KEYMATRIX_F1]))
					{
					gPanelObj.SetPicture = PIC_OVERVIEW;
				}

				gPanelObj.idxKeyPicture[S$KEYMATRIX_F2] = STATE_SUB_PAGE;
					if(1 == EDGEPOS(gPanelObj.KeyMatric[S$KEYMATRIX_F2],KeyMatric[S$KEYMATRIX_F2]))
					{
					gPanelObj.SetPicture = gPanelObj.OldPicture;
				}

				gPanelObj.idxKeyPicture[S$KEYMATRIX_F3] = STATE_SUB_PAGE;
					if(1 == EDGEPOS(gPanelObj.KeyMatric[S$KEYMATRIX_F3],KeyMatric[S$KEYMATRIX_F3]))
					{
					//					if(PIC_IO_DI_1 == gPanelObj.GetPicture)
					//					{
					//						gPanelObj.SetPicture = PIC_IO_DI_2;
					//					}
					//					else
					//					{
					gPanelObj.SetPicture = PIC_IO_DI_1;
					//					}
				}

				if(gPanelObj.GetPicture >= PIC_IO_DI_1 && gPanelObj.GetPicture <= PIC_IO_DI_3)
				{
					gPanelObj.idxKeyPicture[S$KEYMATRIX_F3] = STATE_ACTIVE;
						}

				gPanelObj.idxKeyPicture[S$KEYMATRIX_F4] = STATE_SUB_PAGE;
					if(1 == EDGEPOS(gPanelObj.KeyMatric[S$KEYMATRIX_F4],KeyMatric[S$KEYMATRIX_F4]))
					{
					gPanelObj.SetPicture = PIC_IO_DO_1;
				}

				gPanelObj.idxKeyPicture[S$KEYMATRIX_F5] = STATE_SUB_PAGE;
					if(1 == EDGEPOS(gPanelObj.KeyMatric[S$KEYMATRIX_F5],KeyMatric[S$KEYMATRIX_F5]))
					{
					gPanelObj.SetPicture = PIC_IO_AI_1;
				}
				if(gPanelObj.GetPicture == PIC_IO_AI_1)
				{
					gPanelObj.idxKeyPicture[S$KEYMATRIX_F5] = STATE_ACTIVE;
						}

				gPanelObj.idxKeyPicture[S$KEYMATRIX_F6] = STATE_SUB_PAGE;
					if(1 == EDGEPOS(gPanelObj.KeyMatric[S$KEYMATRIX_F6],KeyMatric[S$KEYMATRIX_F6]))
					{
					gPanelObj.SetPicture = PIC_IO_AO_1;
				}

				gPanelObj.idxKeyPicture[S$KEYMATRIX_F7] = STATE_SUB_PAGE;
					if(1 == EDGEPOS(gPanelObj.KeyMatric[S$KEYMATRIX_F7],KeyMatric[S$KEYMATRIX_F7]))
					{
					gPanelObj.SetPicture = PIC_IO_MODULE;
				}
				if(gPanelObj.GetPicture == PIC_IO_MODULE)
				{
					gPanelObj.idxKeyPicture[S$KEYMATRIX_F7] = STATE_ACTIVE;
						}

				gPanelObj.idxKeyPicture[S$KEYMATRIX_F8]  = STATE_INACTIVE;
					gPanelObj.idxKeyPicture[S$KEYMATRIX_F9]  = STATE_INACTIVE;

					if (gPanelObj.PasswordLevel <= 3)
				{
					gPanelObj.idxKeyPicture[S$KEYMATRIX_F10] = STATE_INACTIVE;
						}
				else
				{
					if(1 == EDGEPOS(gPanelObj.KeyMatric[S$KEYMATRIX_F10],KeyMatric[S$KEYMATRIX_F10]))
						{
						gPanelObj.SetPicture = PIC_MOTOR_TREND;
					}
				}
				//						gPanelObj.idxKeyPicture[S$KEYMATRIX_F10] = STATE_INACTIVE;
				gPanelObj.idxKeyPicture[S$KEYMATRIX_F11] = STATE_INACTIVE;
					gPanelObj.idxKeyPicture[S$KEYMATRIX_F12] = STATE_INACTIVE;
					gPanelObj.idxKeyPicture[S$KEYMATRIX_F13] = STATE_INACTIVE;
					gPanelObj.idxKeyPicture[S$KEYMATRIX_F14] = STATE_INACTIVE;
					//						gPanelObj.idxKeyPicture[S$KEYMATRIX_F14] = STATE_SUB_PAGE;
					//						if(1 == EDGEPOS(gPanelObj.KeyMatric[S$KEYMATRIX_F14],KeyMatric[S$KEYMATRIX_F14]))
					//						{
					//						if(gPanelObj.GetPicture != PIC_ENERGY_MONITOR_ALL)
					//						{
					//							gPanelObj.SetPicture = PIC_ENERGY_MONITOR_ALL;
					//						}
					//						else
					//						{
					//							gPanelObj.SetPicture = PIC_ENERGY_MONITOR;
					//						}
					//					}
					//					if(gPanelObj.GetPicture == PIC_ENERGY_MONITOR)gPanelObj.idxKeyPicture[S$KEYMATRIX_F14] = STATE_ACTIVE;

					gPanelObj.idxKeyPicture[S$KEYMATRIX_F15] = STATE_INACTIVE;

					gPanelObj.idxKeyPicture[S$KEYMATRIX_F16] = STATE_SUB_PAGE;
					if(1 == EDGEPOS(gPanelObj.KeyMatric[S$KEYMATRIX_F16],KeyMatric[S$KEYMATRIX_F16]))
					{
					gPanelObj.SetPicture = PIC_PASSWORD_LOGIN;
				}
				break;

			//				case PIC_MOTOR_TREND:
			//					if(ChangePageDly > 0)
			//					{
			//						ChangePageDly--;
			//						break;
			//					}
			//
			//					gPanelObj.idxKeyPicture[S$KEYMATRIX_F1] = STATE_SUB_PAGE;
			//						if(1 == EDGEPOS(gPanelObj.KeyMatric[S$KEYMATRIX_F1],KeyMatric[S$KEYMATRIX_F1]))
			//						{
			//						gPanelObj.SetPicture = PIC_OVERVIEW;
			//					}
			//
			//					gPanelObj.idxKeyPicture[S$KEYMATRIX_F2] = STATE_SUB_PAGE;
			//						if(1 == EDGEPOS(gPanelObj.KeyMatric[S$KEYMATRIX_F2],KeyMatric[S$KEYMATRIX_F2]))
			//						{
			//						gPanelObj.SetPicture = gPanelObj.OldPicture;
			//					}
			//
			//					gPanelObj.idxKeyPicture[S$KEYMATRIX_F3] = STATE_SUB_PAGE;
			//						if(1 == EDGEPOS(gPanelObj.KeyMatric[S$KEYMATRIX_F3],KeyMatric[S$KEYMATRIX_F3]))
			//						{
			//						gPanelObj.SetPicture = PIC_IO_DI_1;
			//						//						if(PIC_IO_DI_1==gPanelObj.GetPicture)
			//						//						{
			//						//							gPanelObj.SetPicture = PIC_IO_DI_2;
			//						//						}
			//						//						else
			//						//						{
			//						//							gPanelObj.SetPicture = PIC_IO_DI_1;
			//						//						}
			//					}
			//
			//
			//					if(gPanelObj.GetPicture >= PIC_IO_DI_1 && gPanelObj.GetPicture <= PIC_IO_DI_3)
			//					{
			//						gPanelObj.idxKeyPicture[S$KEYMATRIX_F3] = STATE_ACTIVE;
			//							}
			//
			//					gPanelObj.idxKeyPicture[S$KEYMATRIX_F4] = STATE_SUB_PAGE;
			//						if(1 == EDGEPOS(gPanelObj.KeyMatric[S$KEYMATRIX_F4],KeyMatric[S$KEYMATRIX_F4]))
			//						{
			//						gPanelObj.SetPicture = PIC_IO_DO_1;
			//					}
			//
			//					gPanelObj.idxKeyPicture[S$KEYMATRIX_F5] = STATE_SUB_PAGE;
			//						if(1 == EDGEPOS(gPanelObj.KeyMatric[S$KEYMATRIX_F5],KeyMatric[S$KEYMATRIX_F5]))
			//						{
			//						gPanelObj.SetPicture = PIC_IO_AI_1;
			//					}
			//					if(gPanelObj.GetPicture == PIC_IO_AI_1)
			//					{
			//						gPanelObj.idxKeyPicture[S$KEYMATRIX_F5] = STATE_ACTIVE;
			//							}
			//
			//					gPanelObj.idxKeyPicture[S$KEYMATRIX_F6] = STATE_SUB_PAGE;
			//						if(1 == EDGEPOS(gPanelObj.KeyMatric[S$KEYMATRIX_F6],KeyMatric[S$KEYMATRIX_F6]))
			//						{
			//						gPanelObj.SetPicture = PIC_IO_AO_1;
			//					}
			//
			//					gPanelObj.idxKeyPicture[S$KEYMATRIX_F7] = STATE_SUB_PAGE;
			//						if(1 == EDGEPOS(gPanelObj.KeyMatric[S$KEYMATRIX_F7],KeyMatric[S$KEYMATRIX_F7]))
			//						{
			//						gPanelObj.SetPicture = PIC_IO_MODULE;
			//					}
			//					if(gPanelObj.GetPicture == PIC_IO_MODULE)
			//					{
			//						gPanelObj.idxKeyPicture[S$KEYMATRIX_F7] = STATE_ACTIVE;
			//							}
			//
			//					gPanelObj.idxKeyPicture[S$KEYMATRIX_F8]  = STATE_INACTIVE;
			//						gPanelObj.idxKeyPicture[S$KEYMATRIX_F9]  = STATE_INACTIVE;
			//
			//						if (gPanelObj.PasswordLevel <= 3)
			//					{
			//						gPanelObj.idxKeyPicture[S$KEYMATRIX_F10] = STATE_INACTIVE;
			//							}
			//					else
			//					{
			//						if(1 == EDGEPOS(gPanelObj.KeyMatric[S$KEYMATRIX_F10],KeyMatric[S$KEYMATRIX_F10]))
			//							{
			//							gPanelObj.SetPicture = PIC_MOTOR_TREND;
			//						}
			//					}
			//					//						gPanelObj.idxKeyPicture[S$KEYMATRIX_F10] = STATE_INACTIVE;
			//					gPanelObj.idxKeyPicture[S$KEYMATRIX_F11] = STATE_INACTIVE;
			//						gPanelObj.idxKeyPicture[S$KEYMATRIX_F12] = STATE_INACTIVE;
			//						gPanelObj.idxKeyPicture[S$KEYMATRIX_F13] = STATE_INACTIVE;
			//						gPanelObj.idxKeyPicture[S$KEYMATRIX_F14] = STATE_INACTIVE;
			//						//						gPanelObj.idxKeyPicture[S$KEYMATRIX_F14] = STATE_SUB_PAGE;
			//						//						if(1 == EDGEPOS(gPanelObj.KeyMatric[S$KEYMATRIX_F14],KeyMatric[S$KEYMATRIX_F14]))
			//						//						{
			//						//						if(gPanelObj.GetPicture != PIC_ENERGY_MONITOR_ALL)
			//						//						{
			//						//							gPanelObj.SetPicture = PIC_ENERGY_MONITOR_ALL;
			//						//						}
			//						//						else
			//						//						{
			//						//							gPanelObj.SetPicture = PIC_ENERGY_MONITOR;
			//						//						}
			//						//					}
			//						//					if(gPanelObj.GetPicture == PIC_ENERGY_MONITOR)gPanelObj.idxKeyPicture[S$KEYMATRIX_F14] = STATE_ACTIVE;
			//
			//						gPanelObj.idxKeyPicture[S$KEYMATRIX_F15] = STATE_INACTIVE;
			//
			//						gPanelObj.idxKeyPicture[S$KEYMATRIX_F16] = STATE_SUB_PAGE;
			//						if(1 == EDGEPOS(gPanelObj.KeyMatric[S$KEYMATRIX_F16],KeyMatric[S$KEYMATRIX_F16]))
			//						{
			//						gPanelObj.SetPicture = PIC_PASSWORD_LOGIN;
			//					}
			//					break;
			//				case PIC_AUTO_START:
			//				case PIC_AUTO_STEP:
			//					if(ChangePageDly > 0)
			//					{
			//						ChangePageDly--;
			//						break;
			//					}
			//
			//					gPanelObj.idxKeyPicture[S$KEYMATRIX_F1] = STATE_SUB_PAGE;
			//						if(1 == EDGEPOS(gPanelObj.KeyMatric[S$KEYMATRIX_F1],KeyMatric[S$KEYMATRIX_F1]))
			//						{
			//						gPanelObj.SetPicture = PIC_OVERVIEW;
			//					}
			//
			//					gPanelObj.idxKeyPicture[S$KEYMATRIX_F2] = STATE_SUB_PAGE;
			//						if(1 == EDGEPOS(gPanelObj.KeyMatric[S$KEYMATRIX_F2],KeyMatric[S$KEYMATRIX_F2]))
			//						{
			//						gPanelObj.SetPicture = gPanelObj.OldPicture;
			//					}
			//
			//					gPanelObj.idxKeyPicture[S$KEYMATRIX_F3] = STATE_SUB_PAGE;
			//						if(1 == EDGEPOS(gPanelObj.KeyMatric[S$KEYMATRIX_F3],KeyMatric[S$KEYMATRIX_F3]))
			//						{
			//						gPanelObj.SetPicture = PIC_IO_DI_1;
			//					}
			//
			//					gPanelObj.idxKeyPicture[S$KEYMATRIX_F4] = STATE_SUB_PAGE;
			//						if(1 == EDGEPOS(gPanelObj.KeyMatric[S$KEYMATRIX_F4],KeyMatric[S$KEYMATRIX_F4]))
			//						{
			//						gPanelObj.SetPicture = PIC_IO_DO_1;
			//					}
			//
			//					gPanelObj.idxKeyPicture[S$KEYMATRIX_F5] = STATE_SUB_PAGE;
			//						if(1 == EDGEPOS(gPanelObj.KeyMatric[S$KEYMATRIX_F5],KeyMatric[S$KEYMATRIX_F5]))
			//						{
			//						gPanelObj.SetPicture = PIC_IO_AI_1;
			//					}
			//
			//					gPanelObj.idxKeyPicture[S$KEYMATRIX_F6] = STATE_SUB_PAGE;
			//						if(1 == EDGEPOS(gPanelObj.KeyMatric[S$KEYMATRIX_F6],KeyMatric[S$KEYMATRIX_F6]))
			//						{
			//						gPanelObj.SetPicture = PIC_IO_AO_1;
			//					}
			//
			//					gPanelObj.idxKeyPicture[S$KEYMATRIX_F7] = STATE_SUB_PAGE;
			//						if(1 == EDGEPOS(gPanelObj.KeyMatric[S$KEYMATRIX_F7],KeyMatric[S$KEYMATRIX_F7]))
			//						{
			//						gPanelObj.SetPicture = PIC_IO_MODULE;
			//					}
			//
			//					gPanelObj.idxKeyPicture[S$KEYMATRIX_F8]  = STATE_INACTIVE;
			//						gPanelObj.idxKeyPicture[S$KEYMATRIX_F9]  = STATE_INACTIVE;
			//						gPanelObj.idxKeyPicture[S$KEYMATRIX_F10] = STATE_INACTIVE;
			//						gPanelObj.idxKeyPicture[S$KEYMATRIX_F11] = STATE_INACTIVE;
			//						gPanelObj.idxKeyPicture[S$KEYMATRIX_F12] = STATE_INACTIVE;
			//						gPanelObj.idxKeyPicture[S$KEYMATRIX_F13] = STATE_SUB_PAGE;
			//
			//						if(1 == EDGEPOS(gPanelObj.KeyMatric[S$KEYMATRIX_F13],KeyMatric[S$KEYMATRIX_F13]))
			//						{
			//						gPanelObj.SetPicture = PIC_AUTO_STEP;
			//					}
			//					if(gPanelObj.GetPicture == PIC_AUTO_STEP)gPanelObj.idxKeyPicture[S$KEYMATRIX_F13] = STATE_ACTIVE;
			//
			//						gPanelObj.idxKeyPicture[S$KEYMATRIX_F14] = STATE_SUB_PAGE;
			//						if(1 == EDGEPOS(gPanelObj.KeyMatric[S$KEYMATRIX_F14],KeyMatric[S$KEYMATRIX_F14]))
			//						{
			//						gPanelObj.SetPicture = PIC_AUTO_START;
			//					}
			//					if(gPanelObj.GetPicture == PIC_AUTO_START)gPanelObj.idxKeyPicture[S$KEYMATRIX_F14] = STATE_ACTIVE;
			//
			//						gPanelObj.idxKeyPicture[S$KEYMATRIX_F15] = STATE_INACTIVE;
			//
			//						gPanelObj.idxKeyPicture[S$KEYMATRIX_F16] = STATE_SUB_PAGE;
			//						if(1 == EDGEPOS(gPanelObj.KeyMatric[S$KEYMATRIX_F16],KeyMatric[S$KEYMATRIX_F16]))
			//						{
			//						gPanelObj.SetPicture = PIC_PASSWORD_LOGIN;
			//					}
			//					break;

			case PIC_IO_AO_1:			/*  AO FORCE   */
				if(ChangePageDly > 0)
				{
					ChangePageDly--;
					break;
				}

				gPanelObj.idxKeyPicture[S$KEYMATRIX_F1] = STATE_SUB_PAGE;
					if(1 == EDGEPOS(gPanelObj.KeyMatric[S$KEYMATRIX_F1],KeyMatric[S$KEYMATRIX_F1]))
					{
					gPanelObj.SetPicture = PIC_OVERVIEW;
				}

				gPanelObj.idxKeyPicture[S$KEYMATRIX_F2] = STATE_SUB_PAGE;
					if(1 == EDGEPOS(gPanelObj.KeyMatric[S$KEYMATRIX_F2],KeyMatric[S$KEYMATRIX_F2]))
					{
					gPanelObj.SetPicture = gPanelObj.OldPicture;
				}

				gPanelObj.idxKeyPicture[S$KEYMATRIX_F3] = STATE_SUB_PAGE;
					if(1 == EDGEPOS(gPanelObj.KeyMatric[S$KEYMATRIX_F3],KeyMatric[S$KEYMATRIX_F3]))
					{
					gPanelObj.SetPicture = PIC_IO_DI_1;
				}

				gPanelObj.idxKeyPicture[S$KEYMATRIX_F4] = STATE_SUB_PAGE;
					if(1 == EDGEPOS(gPanelObj.KeyMatric[S$KEYMATRIX_F4],KeyMatric[S$KEYMATRIX_F4]))
					{
					gPanelObj.SetPicture = PIC_IO_DO_1;
				}

				gPanelObj.idxKeyPicture[S$KEYMATRIX_F5] = STATE_SUB_PAGE;
					if(1 == EDGEPOS(gPanelObj.KeyMatric[S$KEYMATRIX_F5],KeyMatric[S$KEYMATRIX_F5]))
					{
					gPanelObj.SetPicture = PIC_IO_AI_1;
				}

				gPanelObj.idxKeyPicture[S$KEYMATRIX_F6] = STATE_ACTIVE;
					if(1 == EDGEPOS(gPanelObj.KeyMatric[S$KEYMATRIX_F6],KeyMatric[S$KEYMATRIX_F6]))
					{
					gPanelObj.SetPicture = PIC_IO_AO_1;
				}

				gPanelObj.idxKeyPicture[S$KEYMATRIX_F7] = STATE_SUB_PAGE;
					if(1 == EDGEPOS(gPanelObj.KeyMatric[S$KEYMATRIX_F7],KeyMatric[S$KEYMATRIX_F7]))
					{
					gPanelObj.SetPicture = PIC_IO_MODULE;
				}

				gPanelObj.idxKeyPicture[S$KEYMATRIX_F8] = STATE_INACTIVE;

					if(1 == EDGEPOS(gPanelObj.KeyMatric[S$KEYMATRIX_UP],KeyMatric[S$KEYMATRIX_UP])) /* UP ARROW  */
					{
					if(0 == IndexAo)
					{
						IndexAo = 3;
					}
					else
					{
						IndexAo = IndexAo-1;
					}
				}

				if(1 == EDGEPOS(gPanelObj.KeyMatric[S$KEYMATRIX_DOWN],KeyMatric[S$KEYMATRIX_DOWN])) /* DOWN ARROW  */
					{
					if(3 == IndexAo)
					{
						IndexAo = 0;
					}
					else
					{
						IndexAo = IndexAo+1;
					}
				}

				if(IndexAo > 3)IndexAo = 3;
				if(IndexAo < 0)IndexAo = 0;

				for(i=0;i<4;i++)
				{
					AoColor[i] = 0x00FA;
				}
				if(1 == gTKcalib.Status && gPanelObj.PasswordLevel > 2)
				{
					gPanelObj.idxKeyPicture[S$KEYMATRIX_F9] = STATE_SUB_BUTTON;
						bHideForceAO = 0;
					AoColor[IndexAo] = 0x22A9;
					if(1 == EDGENEG(gPanelObj.KeyMatric[S$KEYMATRIX_F9],KeyMatric[S$KEYMATRIX_F9]))
						{
						if(gHardWare.AOForceNum > 3)
						{
							gHardWare.AOForceNum = IndexAo;
							gImply.ForceAO = 1;
						}
						else
						{
							gHardWare.AOForceNum = 19;
							gImply.ForceAO = 0;
						}

						//							gHardWare.AOForceNum[IndexAo] = !gHardWare.AOForceNum[IndexAo];

					}
				}
				else
				{
					gPanelObj.idxKeyPicture[S$KEYMATRIX_F9] = STATE_INACTIVE;
						bHideForceAO = 1;
					gHardWare.AOForceNum = 19;
					if(1 == gImply.ForceAO)gImply.ForceAO = 0;
				}

				if (gPanelObj.PasswordLevel <= 3)
				{
					gPanelObj.idxKeyPicture[S$KEYMATRIX_F10] = STATE_INACTIVE;
						}
				else
				{
					if(1 == EDGEPOS(gPanelObj.KeyMatric[S$KEYMATRIX_F10],KeyMatric[S$KEYMATRIX_F10]))
						{
						gPanelObj.SetPicture = PIC_MOTOR_TREND;
					}
				}
				//						gPanelObj.idxKeyPicture[S$KEYMATRIX_F10] = STATE_INACTIVE;
				gPanelObj.idxKeyPicture[S$KEYMATRIX_F11] = STATE_INACTIVE;
					gPanelObj.idxKeyPicture[S$KEYMATRIX_F12] = STATE_INACTIVE;
					gPanelObj.idxKeyPicture[S$KEYMATRIX_F13] = STATE_INACTIVE;
					gPanelObj.idxKeyPicture[S$KEYMATRIX_F14] = STATE_INACTIVE;
					//						gPanelObj.idxKeyPicture[S$KEYMATRIX_F14] = STATE_SUB_PAGE;
					//						if(1 == EDGEPOS(gPanelObj.KeyMatric[S$KEYMATRIX_F14],KeyMatric[S$KEYMATRIX_F14]))
					//						{
					//						gPanelObj.SetPicture = PIC_ENERGY_MONITOR;
					//					}
					//					if(gPanelObj.SetPicture == PIC_ENERGY_MONITOR)gPanelObj.idxKeyPicture[S$KEYMATRIX_F14] = STATE_ACTIVE;
					gPanelObj.idxKeyPicture[S$KEYMATRIX_F15] = STATE_INACTIVE;

					gPanelObj.idxKeyPicture[S$KEYMATRIX_F16] = STATE_SUB_PAGE;
					if(1 == EDGEPOS(gPanelObj.KeyMatric[S$KEYMATRIX_F16],KeyMatric[S$KEYMATRIX_F16]))
					{
					gPanelObj.SetPicture = PIC_PASSWORD_LOGIN;
				}
				break;

			case PIC_IO_DO_1:			/*  DO FORCE   */
				if(ChangePageDly > 0)
				{
					ChangePageDly--;
					break;
				}

				gPanelObj.idxKeyPicture[S$KEYMATRIX_F1] = STATE_SUB_PAGE;
					if(1 == EDGEPOS(gPanelObj.KeyMatric[S$KEYMATRIX_F1],KeyMatric[S$KEYMATRIX_F1]))
					{
					gPanelObj.SetPicture = PIC_OVERVIEW;
				}

				gPanelObj.idxKeyPicture[S$KEYMATRIX_F2] = STATE_SUB_PAGE;
					if(1 == EDGEPOS(gPanelObj.KeyMatric[S$KEYMATRIX_F2],KeyMatric[S$KEYMATRIX_F2]))
					{
					gPanelObj.SetPicture = gPanelObj.OldPicture;
				}

				gPanelObj.idxKeyPicture[S$KEYMATRIX_F3] = STATE_SUB_PAGE;
					if(1 == EDGEPOS(gPanelObj.KeyMatric[S$KEYMATRIX_F3],KeyMatric[S$KEYMATRIX_F3]))
					{
					gPanelObj.SetPicture = PIC_IO_DI_1;
				}

				gPanelObj.idxKeyPicture[S$KEYMATRIX_F4] = STATE_ACTIVE;
					if(1 == EDGEPOS(gPanelObj.KeyMatric[S$KEYMATRIX_F4],KeyMatric[S$KEYMATRIX_F4]))
					{
					gPanelObj.SetPicture = PIC_IO_DO_3;
				}

				gPanelObj.idxKeyPicture[S$KEYMATRIX_F5] = STATE_SUB_PAGE;
					if(1 == EDGEPOS(gPanelObj.KeyMatric[S$KEYMATRIX_F5],KeyMatric[S$KEYMATRIX_F5]))
					{
					gPanelObj.SetPicture = PIC_IO_AI_1;
				}

				gPanelObj.idxKeyPicture[S$KEYMATRIX_F6] = STATE_SUB_PAGE;
					if(1 == EDGEPOS(gPanelObj.KeyMatric[S$KEYMATRIX_F6],KeyMatric[S$KEYMATRIX_F6]))
					{
					gPanelObj.SetPicture = PIC_IO_AO_1;
				}

				gPanelObj.idxKeyPicture[S$KEYMATRIX_F7] = STATE_SUB_PAGE;
					if(1 == EDGEPOS(gPanelObj.KeyMatric[S$KEYMATRIX_F7],KeyMatric[S$KEYMATRIX_F7]))
					{
					gPanelObj.SetPicture = PIC_IO_MODULE;
				}

				gPanelObj.idxKeyPicture[S$KEYMATRIX_F8] = STATE_INACTIVE;

					if(1 == EDGEPOS(gPanelObj.KeyMatric[S$KEYMATRIX_UP],KeyMatric[S$KEYMATRIX_UP])) 	/* UP ARROW  */
					{
					if(0 == IndexDo)
					{
						IndexDo = MAX_PAGE_DO32 - 1;
					}
					else
					{
						IndexDo = IndexDo-1;
					}
				}

				if(1 == EDGEPOS(gPanelObj.KeyMatric[S$KEYMATRIX_DOWN],KeyMatric[S$KEYMATRIX_DOWN])) /* DOWN ARROW  */
					{
					if(MAX_PAGE_DO48 - 1 == IndexDo)
					{
						IndexDo = 0;
					}
					else
					{
						IndexDo = IndexDo+1;
					}
				}

				if(1 == EDGEPOS(gPanelObj.KeyMatric[S$KEYMATRIX_LEFT],KeyMatric[S$KEYMATRIX_LEFT])) /* LEFT ARROW  */
					{
					IndexDo = IndexDo - 8;
					if(IndexDo < 0)IndexDo = MAX_PAGE_DO32 + IndexDo;
				}

				if(1 == EDGEPOS(gPanelObj.KeyMatric[S$KEYMATRIX_RIGHT],KeyMatric[S$KEYMATRIX_RIGHT])) /* RIGHT ARROW  */
					{
					IndexDo = IndexDo + 8;
					if(IndexDo > MAX_PAGE_DO32 - 1)IndexDo = IndexDo - MAX_PAGE_DO32;
				}

				if(IndexDo > MAX_PAGE_DO32 - 1)IndexDo = MAX_PAGE_DO - 1;
				if(IndexDo < 0 )IndexDo = 0;

				for(i=0;i<MAX_PAGE_DO32;i++)
				{
					DoColor[i] = 0x00FA;
				}

				if(1 == gTKcalib.Status && gPanelObj.PasswordLevel > 2)
				{
					gPanelObj.idxKeyPicture[S$KEYMATRIX_F9] = STATE_SUB_BUTTON;
						DoColor[IndexDo] = 0x22A9;
					if(1 == EDGEPOS(gPanelObj.KeyMatric[S$KEYMATRIX_F9],KeyMatric[S$KEYMATRIX_F9]))
						{
						gHardWare.DOForce[IndexDo] = !gHardWare.DOForce[IndexDo];
					}
				}
				else
				{
					gPanelObj.idxKeyPicture[S$KEYMATRIX_F9] = STATE_INACTIVE;
						}

				if (gPanelObj.PasswordLevel <= 3)
				{
					gPanelObj.idxKeyPicture[S$KEYMATRIX_F10] = STATE_INACTIVE;
						}
				else
				{
					if(1 == EDGEPOS(gPanelObj.KeyMatric[S$KEYMATRIX_F10],KeyMatric[S$KEYMATRIX_F10]))
						{
						gPanelObj.SetPicture = PIC_MOTOR_TREND;
					}
				}
				//						gPanelObj.idxKeyPicture[S$KEYMATRIX_F10] = STATE_INACTIVE;
				gPanelObj.idxKeyPicture[S$KEYMATRIX_F11] = STATE_INACTIVE;
					gPanelObj.idxKeyPicture[S$KEYMATRIX_F12] = STATE_INACTIVE;
					gPanelObj.idxKeyPicture[S$KEYMATRIX_F13] = STATE_INACTIVE;
					gPanelObj.idxKeyPicture[S$KEYMATRIX_F14] = STATE_INACTIVE;
					//						gPanelObj.idxKeyPicture[S$KEYMATRIX_F14] = STATE_SUB_PAGE;
					//						if(1 == EDGEPOS(gPanelObj.KeyMatric[S$KEYMATRIX_F14],KeyMatric[S$KEYMATRIX_F14]))
					//						{
					//						gPanelObj.SetPicture = PIC_ENERGY_MONITOR;
					//					}
					//					if(gPanelObj.SetPicture == PIC_ENERGY_MONITOR)gPanelObj.idxKeyPicture[S$KEYMATRIX_F14] = STATE_ACTIVE;
					gPanelObj.idxKeyPicture[S$KEYMATRIX_F15] = STATE_INACTIVE;

					gPanelObj.idxKeyPicture[S$KEYMATRIX_F16] = STATE_SUB_PAGE;
					if(1 == EDGEPOS(gPanelObj.KeyMatric[S$KEYMATRIX_F16],KeyMatric[S$KEYMATRIX_F16]))
					{
					gPanelObj.SetPicture = PIC_PASSWORD_LOGIN;
				}
				break;

			case PIC_IO_DO_2:
				if(ChangePageDly > 0)
				{
					ChangePageDly--;
					break;
				}

				gPanelObj.idxKeyPicture[S$KEYMATRIX_F1] = STATE_SUB_PAGE;
					if(1 == EDGEPOS(gPanelObj.KeyMatric[S$KEYMATRIX_F1],KeyMatric[S$KEYMATRIX_F1]))
					{
					gPanelObj.SetPicture = PIC_OVERVIEW;
				}

				gPanelObj.idxKeyPicture[S$KEYMATRIX_F2] = STATE_SUB_PAGE;
					if(1 == EDGEPOS(gPanelObj.KeyMatric[S$KEYMATRIX_F2],KeyMatric[S$KEYMATRIX_F2]))
					{
					gPanelObj.SetPicture = gPanelObj.OldPicture;
				}

				gPanelObj.idxKeyPicture[S$KEYMATRIX_F3] = STATE_SUB_PAGE;
					if(1 == EDGEPOS(gPanelObj.KeyMatric[S$KEYMATRIX_F3],KeyMatric[S$KEYMATRIX_F3]))
					{
					gPanelObj.SetPicture = PIC_IO_DI_1;
				}

				gPanelObj.idxKeyPicture[S$KEYMATRIX_F4] = STATE_ACTIVE;
					if(1 == EDGEPOS(gPanelObj.KeyMatric[S$KEYMATRIX_F4],KeyMatric[S$KEYMATRIX_F4]))
					{
					gPanelObj.SetPicture = PIC_IO_DO_3;
				}

				gPanelObj.idxKeyPicture[S$KEYMATRIX_F5] = STATE_SUB_PAGE;
					if(1 == EDGEPOS(gPanelObj.KeyMatric[S$KEYMATRIX_F5],KeyMatric[S$KEYMATRIX_F5]))
					{
					gPanelObj.SetPicture = PIC_IO_AI_1;
				}

				gPanelObj.idxKeyPicture[S$KEYMATRIX_F6] = STATE_SUB_PAGE;
					if(1 == EDGEPOS(gPanelObj.KeyMatric[S$KEYMATRIX_F6],KeyMatric[S$KEYMATRIX_F6]))
					{
					gPanelObj.SetPicture = PIC_IO_AO_1;
				}

				gPanelObj.idxKeyPicture[S$KEYMATRIX_F7] = STATE_SUB_PAGE;
					if(1 == EDGEPOS(gPanelObj.KeyMatric[S$KEYMATRIX_F7],KeyMatric[S$KEYMATRIX_F7]))
					{
					gPanelObj.SetPicture = PIC_IO_MODULE;
				}

				gPanelObj.idxKeyPicture[S$KEYMATRIX_F8] = STATE_INACTIVE;

					if(1 == EDGEPOS(gPanelObj.KeyMatric[S$KEYMATRIX_UP],KeyMatric[S$KEYMATRIX_UP])) 	/* UP ARROW  */
					{
					if(0 == IndexDo)
					{
						IndexDo = MAX_PAGE_DO - 1;
					}
					else
					{
						IndexDo = IndexDo-1;
					}
				}

				if(1 == EDGEPOS(gPanelObj.KeyMatric[S$KEYMATRIX_DOWN],KeyMatric[S$KEYMATRIX_DOWN])) /* DOWN ARROW  */
					{
					if(MAX_PAGE_DO - 1 == IndexDo)
					{
						IndexDo = 0;
					}
					else
					{
						IndexDo = IndexDo+1;
					}
				}

				if(1 == EDGEPOS(gPanelObj.KeyMatric[S$KEYMATRIX_LEFT],KeyMatric[S$KEYMATRIX_LEFT])) /* LEFT ARROW  */
					{
					IndexDo = IndexDo - 16;
					if(IndexDo < 0)IndexDo = MAX_PAGE_DO + IndexDo;
				}

				if(1 == EDGEPOS(gPanelObj.KeyMatric[S$KEYMATRIX_RIGHT],KeyMatric[S$KEYMATRIX_RIGHT])) /* RIGHT ARROW  */
					{
					IndexDo = IndexDo + 16;
					if(IndexDo > MAX_PAGE_DO - 1)IndexDo = IndexDo - MAX_PAGE_DO;
				}

				if(IndexDo > MAX_PAGE_DO - 1)IndexDo = MAX_PAGE_DO - 1;
				if(IndexDo < 0 )IndexDo = 0;

				for(i=0;i<MAX_PAGE_DO;i++)
				{
					DoColor[i + MAX_PAGE_DO] = 0x00FA;
				}

				if(1 == gTKcalib.Status && gPanelObj.PasswordLevel > 2)
				{
					gPanelObj.idxKeyPicture[S$KEYMATRIX_F9] = STATE_SUB_BUTTON;
						DoColor[IndexDo + MAX_PAGE_DO] = 0x22A9;
					if(1 == EDGENEG(gPanelObj.KeyMatric[S$KEYMATRIX_F9],KeyMatric[S$KEYMATRIX_F9]))
						{
						gHardWare.DOForce[IndexDo + MAX_PAGE_DO] = !gHardWare.DOForce[IndexDo + MAX_PAGE_DO];
					}
				}
				else
				{
					gPanelObj.idxKeyPicture[S$KEYMATRIX_F9] = STATE_INACTIVE;
						}

				if (gPanelObj.PasswordLevel <= 3)
				{
					gPanelObj.idxKeyPicture[S$KEYMATRIX_F10] = STATE_INACTIVE;
						}
				else
				{
					if(1 == EDGEPOS(gPanelObj.KeyMatric[S$KEYMATRIX_F10],KeyMatric[S$KEYMATRIX_F10]))
						{
						gPanelObj.SetPicture = PIC_MOTOR_TREND;
					}
				}
				//						gPanelObj.idxKeyPicture[S$KEYMATRIX_F10] = STATE_INACTIVE;
				gPanelObj.idxKeyPicture[S$KEYMATRIX_F11] = STATE_INACTIVE;
					gPanelObj.idxKeyPicture[S$KEYMATRIX_F12] = STATE_INACTIVE;
					gPanelObj.idxKeyPicture[S$KEYMATRIX_F13] = STATE_INACTIVE;
					gPanelObj.idxKeyPicture[S$KEYMATRIX_F14] = STATE_INACTIVE;
					//						gPanelObj.idxKeyPicture[S$KEYMATRIX_F14] = STATE_SUB_PAGE;
					//						if(1 == EDGEPOS(gPanelObj.KeyMatric[S$KEYMATRIX_F14],KeyMatric[S$KEYMATRIX_F14]))
					//						{
					//						gPanelObj.SetPicture = PIC_ENERGY_MONITOR;
					//					}
					//					if(gPanelObj.SetPicture == PIC_ENERGY_MONITOR)gPanelObj.idxKeyPicture[S$KEYMATRIX_F14] = STATE_ACTIVE;
					gPanelObj.idxKeyPicture[S$KEYMATRIX_F15] = STATE_INACTIVE;

					gPanelObj.idxKeyPicture[S$KEYMATRIX_F16] = STATE_SUB_PAGE;
					if(1 == EDGEPOS(gPanelObj.KeyMatric[S$KEYMATRIX_F16],KeyMatric[S$KEYMATRIX_F16]))
					{
					gPanelObj.SetPicture = PIC_PASSWORD_LOGIN;
				}
				break;

			case PIC_IO_DO_3:
				if(ChangePageDly > 0)
				{
					ChangePageDly--;
					break;
				}

				gPanelObj.idxKeyPicture[S$KEYMATRIX_F1] = STATE_SUB_PAGE;
					if(1 == EDGEPOS(gPanelObj.KeyMatric[S$KEYMATRIX_F1],KeyMatric[S$KEYMATRIX_F1]))
					{
					gPanelObj.SetPicture = PIC_OVERVIEW;
				}

				gPanelObj.idxKeyPicture[S$KEYMATRIX_F2] = STATE_SUB_PAGE;
					if(1 == EDGEPOS(gPanelObj.KeyMatric[S$KEYMATRIX_F2],KeyMatric[S$KEYMATRIX_F2]))
					{
					gPanelObj.SetPicture = gPanelObj.OldPicture;
				}

				gPanelObj.idxKeyPicture[S$KEYMATRIX_F3] = STATE_SUB_PAGE;
					if(1 == EDGEPOS(gPanelObj.KeyMatric[S$KEYMATRIX_F3],KeyMatric[S$KEYMATRIX_F3]))
					{
					gPanelObj.SetPicture = PIC_IO_DI_1;
				}

				gPanelObj.idxKeyPicture[S$KEYMATRIX_F4] = STATE_ACTIVE;
					if(1 == EDGEPOS(gPanelObj.KeyMatric[S$KEYMATRIX_F4],KeyMatric[S$KEYMATRIX_F4]))
					{
					gPanelObj.SetPicture = PIC_IO_DO_1;
				}

				gPanelObj.idxKeyPicture[S$KEYMATRIX_F5] = STATE_SUB_PAGE;
					if(1 == EDGEPOS(gPanelObj.KeyMatric[S$KEYMATRIX_F5],KeyMatric[S$KEYMATRIX_F5]))
					{
					gPanelObj.SetPicture = PIC_IO_AI_1;
				}

				gPanelObj.idxKeyPicture[S$KEYMATRIX_F6] = STATE_SUB_PAGE;
					if(1 == EDGEPOS(gPanelObj.KeyMatric[S$KEYMATRIX_F6],KeyMatric[S$KEYMATRIX_F6]))
					{
					gPanelObj.SetPicture = PIC_IO_AO_1;
				}

				gPanelObj.idxKeyPicture[S$KEYMATRIX_F7] = STATE_SUB_PAGE;
					if(1 == EDGEPOS(gPanelObj.KeyMatric[S$KEYMATRIX_F7],KeyMatric[S$KEYMATRIX_F7]))
					{
					gPanelObj.SetPicture = PIC_IO_MODULE;
				}

				gPanelObj.idxKeyPicture[S$KEYMATRIX_F8] = STATE_INACTIVE;

					if(1 == EDGEPOS(gPanelObj.KeyMatric[S$KEYMATRIX_UP],KeyMatric[S$KEYMATRIX_UP])) 	/* UP ARROW  */
					{
					if(0 == IndexDo)
					{
						IndexDo = MAX_PAGE_DO48 - 1;
					}
					else
					{
						IndexDo = IndexDo - 1;
					}
				}

				if(1 == EDGEPOS(gPanelObj.KeyMatric[S$KEYMATRIX_DOWN],KeyMatric[S$KEYMATRIX_DOWN])) /* DOWN ARROW  */
					{
					if(MAX_PAGE_DO48 - 1 == IndexDo)
					{
						IndexDo = 0;
					}
					else
					{
						IndexDo = IndexDo+1;
					}
				}

				if(1 == EDGEPOS(gPanelObj.KeyMatric[S$KEYMATRIX_LEFT],KeyMatric[S$KEYMATRIX_LEFT])) /* LEFT ARROW  */
					{
					IndexDo = IndexDo - 16;
					if(IndexDo < 0)IndexDo = MAX_PAGE_DO48 + IndexDo;
				}

				if(1 == EDGEPOS(gPanelObj.KeyMatric[S$KEYMATRIX_RIGHT],KeyMatric[S$KEYMATRIX_RIGHT])) /* RIGHT ARROW  */
					{
					IndexDo = IndexDo + 16;
					if(IndexDo > MAX_PAGE_DO48 - 1)IndexDo = IndexDo - MAX_PAGE_DO48;
				}

				if(IndexDo > MAX_PAGE_DO48 - 1)IndexDo = MAX_PAGE_DO48 - 1;
				if(IndexDo < 0 )IndexDo = 0;

				for(i=0;i<MAX_PAGE_DO48;i++)
				{
					DoColor[i + MAX_PAGE_DO32] = 0x00FA;
				}

				if(1 == gTKcalib.Status && gPanelObj.PasswordLevel > 2)
				{
					gPanelObj.idxKeyPicture[S$KEYMATRIX_F9] = STATE_SUB_BUTTON;
						DoColor[IndexDo + MAX_PAGE_DO32] = 0x22A9;
					if(1 == EDGENEG(gPanelObj.KeyMatric[S$KEYMATRIX_F9],KeyMatric[S$KEYMATRIX_F9]))
						{
						gHardWare.DOForce[IndexDo + MAX_PAGE_DO32] = !gHardWare.DOForce[IndexDo + MAX_PAGE_DO32];
					}
				}
				else
				{
					gPanelObj.idxKeyPicture[S$KEYMATRIX_F9] = STATE_INACTIVE;
						}

				if (gPanelObj.PasswordLevel <= 3)
				{
					gPanelObj.idxKeyPicture[S$KEYMATRIX_F10] = STATE_INACTIVE;
						}
				else
				{
					if(1 == EDGEPOS(gPanelObj.KeyMatric[S$KEYMATRIX_F10],KeyMatric[S$KEYMATRIX_F10]))
						{
						gPanelObj.SetPicture = PIC_MOTOR_TREND;
					}
				}
				//						gPanelObj.idxKeyPicture[S$KEYMATRIX_F10] = STATE_INACTIVE;
				gPanelObj.idxKeyPicture[S$KEYMATRIX_F11] = STATE_INACTIVE;
					gPanelObj.idxKeyPicture[S$KEYMATRIX_F12] = STATE_INACTIVE;
					gPanelObj.idxKeyPicture[S$KEYMATRIX_F13] = STATE_INACTIVE;
					gPanelObj.idxKeyPicture[S$KEYMATRIX_F14] = STATE_INACTIVE;
					//						gPanelObj.idxKeyPicture[S$KEYMATRIX_F14] = STATE_SUB_PAGE;
					//						if(1 == EDGEPOS(gPanelObj.KeyMatric[S$KEYMATRIX_F14],KeyMatric[S$KEYMATRIX_F14]))
					//						{
					//						gPanelObj.SetPicture = PIC_ENERGY_MONITOR;
					//					}
					//					if(gPanelObj.SetPicture == PIC_ENERGY_MONITOR)gPanelObj.idxKeyPicture[S$KEYMATRIX_F14] = STATE_ACTIVE;
					gPanelObj.idxKeyPicture[S$KEYMATRIX_F15] = STATE_INACTIVE;

					gPanelObj.idxKeyPicture[S$KEYMATRIX_F16] = STATE_SUB_PAGE;
					if(1 == EDGEPOS(gPanelObj.KeyMatric[S$KEYMATRIX_F16],KeyMatric[S$KEYMATRIX_F16]))
					{
					gPanelObj.SetPicture = PIC_PASSWORD_LOGIN;
				}
				break;
			case PIC_IO_DO_4:
				if(ChangePageDly > 0)
				{
					ChangePageDly--;
					break;
				}

				gPanelObj.idxKeyPicture[S$KEYMATRIX_F1] = STATE_SUB_PAGE;
					if(1 == EDGEPOS(gPanelObj.KeyMatric[S$KEYMATRIX_F1],KeyMatric[S$KEYMATRIX_F1]))
					{
					gPanelObj.SetPicture = PIC_OVERVIEW;
				}

				gPanelObj.idxKeyPicture[S$KEYMATRIX_F2] = STATE_SUB_PAGE;
					if(1 == EDGEPOS(gPanelObj.KeyMatric[S$KEYMATRIX_F2],KeyMatric[S$KEYMATRIX_F2]))
					{
					gPanelObj.SetPicture = gPanelObj.OldPicture;
				}

				gPanelObj.idxKeyPicture[S$KEYMATRIX_F3] = STATE_SUB_PAGE;
					if(1 == EDGEPOS(gPanelObj.KeyMatric[S$KEYMATRIX_F3],KeyMatric[S$KEYMATRIX_F3]))
					{
					gPanelObj.SetPicture = PIC_IO_DI_1;
				}

				gPanelObj.idxKeyPicture[S$KEYMATRIX_F4] = STATE_ACTIVE;
					if(1 == EDGEPOS(gPanelObj.KeyMatric[S$KEYMATRIX_F4],KeyMatric[S$KEYMATRIX_F4]))
					{
					gPanelObj.SetPicture = PIC_IO_DO_1;
				}

				gPanelObj.idxKeyPicture[S$KEYMATRIX_F5] = STATE_SUB_PAGE;
					if(1 == EDGEPOS(gPanelObj.KeyMatric[S$KEYMATRIX_F5],KeyMatric[S$KEYMATRIX_F5]))
					{
					gPanelObj.SetPicture = PIC_IO_AI_1;
				}

				gPanelObj.idxKeyPicture[S$KEYMATRIX_F6] = STATE_SUB_PAGE;
					if(1 == EDGEPOS(gPanelObj.KeyMatric[S$KEYMATRIX_F6],KeyMatric[S$KEYMATRIX_F6]))
					{
					gPanelObj.SetPicture = PIC_IO_AO_1;
				}

				gPanelObj.idxKeyPicture[S$KEYMATRIX_F7] = STATE_SUB_PAGE;
					if(1 == EDGEPOS(gPanelObj.KeyMatric[S$KEYMATRIX_F7],KeyMatric[S$KEYMATRIX_F7]))
					{
					gPanelObj.SetPicture = PIC_IO_MODULE;
				}

				gPanelObj.idxKeyPicture[S$KEYMATRIX_F8] = STATE_INACTIVE;

					if(1 == EDGEPOS(gPanelObj.KeyMatric[S$KEYMATRIX_UP],KeyMatric[S$KEYMATRIX_UP])) 	/* UP ARROW  */
					{
					if(0 == IndexDo)
					{
						IndexDo = MAX_PAGE_DO - 1;
					}
					else
					{
						IndexDo = IndexDo - 1;
					}
				}

				if(1 == EDGEPOS(gPanelObj.KeyMatric[S$KEYMATRIX_DOWN],KeyMatric[S$KEYMATRIX_DOWN])) /* DOWN ARROW  */
					{
					if(MAX_PAGE_DO - 1 == IndexDo)
					{
						IndexDo = 0;
					}
					else
					{
						IndexDo = IndexDo+1;
					}
				}

				if(1 == EDGEPOS(gPanelObj.KeyMatric[S$KEYMATRIX_LEFT],KeyMatric[S$KEYMATRIX_LEFT])) /* LEFT ARROW  */
					{
					IndexDo = IndexDo - 16;
					if(IndexDo < 0)IndexDo = MAX_PAGE_DO + IndexDo;
				}

				if(1 == EDGEPOS(gPanelObj.KeyMatric[S$KEYMATRIX_RIGHT],KeyMatric[S$KEYMATRIX_RIGHT])) /* RIGHT ARROW  */
					{
					IndexDo = IndexDo + 16;
					if(IndexDo > MAX_PAGE_DO - 1)IndexDo = IndexDo - MAX_PAGE_DO;
				}

				if(IndexDo > MAX_PAGE_DO - 1)IndexDo = MAX_PAGE_DO - 1;
				if(IndexDo < 0 )IndexDo = 0;

				for(i=0;i<MAX_PAGE_DO;i++)
				{
					DoColor[i + MAX_PAGE_DO32 + MAX_PAGE_DO] = 0x00FA;
				}

				if(1 == gTKcalib.Status && gPanelObj.PasswordLevel > 2)
				{
					gPanelObj.idxKeyPicture[S$KEYMATRIX_F9] = STATE_SUB_BUTTON;
						DoColor[IndexDo +MAX_PAGE_DO32 + MAX_PAGE_DO] = 0x22A9;
					if(1 == EDGENEG(gPanelObj.KeyMatric[S$KEYMATRIX_F9],KeyMatric[S$KEYMATRIX_F9]))
						{
						gHardWare.DOForce[IndexDo + MAX_PAGE_DO32 + MAX_PAGE_DO] = !gHardWare.DOForce[IndexDo + MAX_PAGE_DO32 + MAX_PAGE_DO];
					}
				}
				else
				{
					gPanelObj.idxKeyPicture[S$KEYMATRIX_F9] = STATE_INACTIVE;
						}

				if (gPanelObj.PasswordLevel <= 3)
				{
					gPanelObj.idxKeyPicture[S$KEYMATRIX_F10] = STATE_INACTIVE;
						}
				else
				{
					if(1 == EDGEPOS(gPanelObj.KeyMatric[S$KEYMATRIX_F10],KeyMatric[S$KEYMATRIX_F10]))
						{
						gPanelObj.SetPicture = PIC_MOTOR_TREND;
					}
				}
				//						gPanelObj.idxKeyPicture[S$KEYMATRIX_F10] = STATE_INACTIVE;
				gPanelObj.idxKeyPicture[S$KEYMATRIX_F11] = STATE_INACTIVE;
					gPanelObj.idxKeyPicture[S$KEYMATRIX_F12] = STATE_INACTIVE;
					gPanelObj.idxKeyPicture[S$KEYMATRIX_F13] = STATE_INACTIVE;
					gPanelObj.idxKeyPicture[S$KEYMATRIX_F14] = STATE_INACTIVE;
					//						gPanelObj.idxKeyPicture[S$KEYMATRIX_F14] = STATE_SUB_PAGE;
					//						if(1 == EDGEPOS(gPanelObj.KeyMatric[S$KEYMATRIX_F14],KeyMatric[S$KEYMATRIX_F14]))
					//						{
					//						gPanelObj.SetPicture = PIC_ENERGY_MONITOR;
					//					}
					//					if(gPanelObj.SetPicture == PIC_ENERGY_MONITOR)gPanelObj.idxKeyPicture[S$KEYMATRIX_F14] = STATE_ACTIVE;
					gPanelObj.idxKeyPicture[S$KEYMATRIX_F15] = STATE_INACTIVE;

					gPanelObj.idxKeyPicture[S$KEYMATRIX_F16] = STATE_SUB_PAGE;
					if(1 == EDGEPOS(gPanelObj.KeyMatric[S$KEYMATRIX_F16],KeyMatric[S$KEYMATRIX_F16]))
					{
					gPanelObj.SetPicture = PIC_PASSWORD_LOGIN;
				}
				break;
			case PIC_ALARM_CURRENT:
			case PIC_ALARM_HISTORY:
			case PIC_ALARM_1:
			case PIC_ALARM_2:
			case PIC_ALARM_3:
			case PIC_ALARM_4:
			case PIC_ALARM_5:
				if(ChangePageDly > 0)
				{
					ChangePageDly--;
					break;
				}

				gPanelObj.idxKeyPicture[S$KEYMATRIX_F1] = STATE_SUB_PAGE;
					if(1 == EDGEPOS(gPanelObj.KeyMatric[S$KEYMATRIX_F1],KeyMatric[S$KEYMATRIX_F1]))
					{
					gPanelObj.SetPicture = PIC_OVERVIEW;
				}

				gPanelObj.idxKeyPicture[S$KEYMATRIX_F2] = STATE_SUB_PAGE;
					if(1 == EDGEPOS(gPanelObj.KeyMatric[S$KEYMATRIX_F2],KeyMatric[S$KEYMATRIX_F2]))
					{
					gPanelObj.SetPicture = gPanelObj.OldPicture;
				}

				gPanelObj.idxKeyPicture[S$KEYMATRIX_F3] = STATE_SUB_PAGE;
					if(1 == EDGEPOS(gPanelObj.KeyMatric[S$KEYMATRIX_F3],KeyMatric[S$KEYMATRIX_F3]))
					{
					gPanelObj.SetPicture = PIC_ALARM_CURRENT;
				}
				if(gPanelObj.GetPicture == PIC_ALARM_CURRENT)gPanelObj.idxKeyPicture[S$KEYMATRIX_F3] = STATE_ACTIVE;

					gPanelObj.idxKeyPicture[S$KEYMATRIX_F4] = STATE_SUB_PAGE;
					if(1 == EDGEPOS(gPanelObj.KeyMatric[S$KEYMATRIX_F4],KeyMatric[S$KEYMATRIX_F4]))
					{
					gPanelObj.SetPicture = PIC_ALARM_HISTORY;
				}
				if(gPanelObj.GetPicture == PIC_ALARM_HISTORY)gPanelObj.idxKeyPicture[S$KEYMATRIX_F4] = STATE_ACTIVE;

					gPanelObj.idxKeyPicture[S$KEYMATRIX_F5] = STATE_INACTIVE;
					gPanelObj.idxKeyPicture[S$KEYMATRIX_F6] = STATE_INACTIVE;
					gPanelObj.idxKeyPicture[S$KEYMATRIX_F7] = STATE_INACTIVE;
					gPanelObj.idxKeyPicture[S$KEYMATRIX_F8] = STATE_INACTIVE;
					gPanelObj.idxKeyPicture[S$KEYMATRIX_F9] = STATE_INACTIVE;
					gPanelObj.idxKeyPicture[S$KEYMATRIX_F10] = STATE_SUB_BUTTON;
					gPanelObj.idxKeyPicture[S$KEYMATRIX_F11] = STATE_INACTIVE;
					gPanelObj.idxKeyPicture[S$KEYMATRIX_F12] = STATE_INACTIVE;
					gPanelObj.idxKeyPicture[S$KEYMATRIX_F13] = STATE_INACTIVE;
					gPanelObj.idxKeyPicture[S$KEYMATRIX_F14] = STATE_INACTIVE;
					gPanelObj.idxKeyPicture[S$KEYMATRIX_F15] = STATE_INACTIVE;

					gPanelObj.idxKeyPicture[S$KEYMATRIX_F16] = STATE_SUB_PAGE;
					if(1 == EDGEPOS(gPanelObj.KeyMatric[S$KEYMATRIX_F16],KeyMatric[S$KEYMATRIX_F16]))
					{
					gPanelObj.SetPicture = PIC_PASSWORD_LOGIN;
				}
				break;

			case PIC_PASSWORD_LOGIN:
				if(ChangePageDly > 0)
				{
					ChangePageDly--;
					break;
				}

				gPanelObj.idxKeyPicture[S$KEYMATRIX_F1] = STATE_SUB_PAGE;
					if(1 == EDGEPOS(gPanelObj.KeyMatric[S$KEYMATRIX_F1],KeyMatric[S$KEYMATRIX_F1]))
					{
					gPanelObj.SetPicture = PIC_OVERVIEW;
				}

				gPanelObj.idxKeyPicture[S$KEYMATRIX_F2] = STATE_SUB_PAGE;
					if(1 == EDGEPOS(gPanelObj.KeyMatric[S$KEYMATRIX_F2],KeyMatric[S$KEYMATRIX_F2]))
					{
					gPanelObj.SetPicture = gPanelObj.OldPicture;
				}

				gPanelObj.idxKeyPicture[S$KEYMATRIX_F3] = STATE_SUB_PAGE;
					if(1 == EDGEPOS(gPanelObj.KeyMatric[S$KEYMATRIX_F3],KeyMatric[S$KEYMATRIX_F3]))
					{
					if(gPanelObj.PasswordLevel > 2)gPanelObj.SetPicture = PIC_SYSTEM_SET_1 ;
				}
				if(gPanelObj.PasswordLevel <= 2)gPanelObj.idxKeyPicture[S$KEYMATRIX_F3] = STATE_INACTIVE;

					gPanelObj.idxKeyPicture[S$KEYMATRIX_F4] = STATE_SUB_PAGE;
					if(1 == EDGEPOS(gPanelObj.KeyMatric[S$KEYMATRIX_F4],KeyMatric[S$KEYMATRIX_F4]))
					{
					gPanelObj.SetPicture = PIC_ACCU_SETTING ;
				}
				if(gPanelObj.PasswordLevel <= 2)gPanelObj.idxKeyPicture[S$KEYMATRIX_F4] = STATE_INACTIVE;

					gPanelObj.idxKeyPicture[S$KEYMATRIX_F5] = STATE_SUB_PAGE;
					if(1 == EDGEPOS(gPanelObj.KeyMatric[S$KEYMATRIX_F5],KeyMatric[S$KEYMATRIX_F5]))
					{
					if(gPanelObj.PasswordLevel > 3 )gPanelObj.SetPicture = PIC_OEM_SETTING_1;
				}
				if(gPanelObj.PasswordLevel <= 3 )gPanelObj.idxKeyPicture[S$KEYMATRIX_F5] = STATE_INACTIVE;

					gPanelObj.idxKeyPicture[S$KEYMATRIX_F6] = STATE_SUB_PAGE;
					if(1 == EDGEPOS(gPanelObj.KeyMatric[S$KEYMATRIX_F6],KeyMatric[S$KEYMATRIX_F6]))
					{
					if(gPanelObj.PasswordLevel > 0)gPanelObj.SetPicture = PIC_PASSWORD_SET;
				}
				if(gPanelObj.PasswordLevel < 1)gPanelObj.idxKeyPicture[S$KEYMATRIX_F6] = STATE_INACTIVE;
					/*Chaoi*/
					gPanelObj.idxKeyPicture[S$KEYMATRIX_F7] = STATE_SUB_PAGE;
					if(1 == EDGEPOS(gPanelObj.KeyMatric[S$KEYMATRIX_F7],KeyMatric[S$KEYMATRIX_F7]))
					{
					if(gPanelObj.PasswordLevel > 2)gPanelObj.SetPicture = PIC_PRESSURE_CALIBRATION ;
				}
				if(gPanelObj.PasswordLevel <= 2)gPanelObj.idxKeyPicture[S$KEYMATRIX_F7] = STATE_INACTIVE;
					//				gPanelObj.idxKeyPicture[S$KEYMATRIX_F7] = STATE_SUB_PAGE;
					//				if(1 == EDGEPOS(gPanelObj.KeyMatric[S$KEYMATRIX_F7],KeyMatric[S$KEYMATRIX_F7]))
					//				{
					//					if(0 == bLevel3CalibHide)
					//					{
					//						gPanelObj.SetPicture = PIC_MOLD_CALIBRATION;
					//					}
					//				}
					//				if(1 == bLevel3CalibHide)gPanelObj.idxKeyPicture[S$KEYMATRIX_F7] = STATE_INACTIVE;

					gPanelObj.idxKeyPicture[S$KEYMATRIX_F8] = STATE_SUB_PAGE;
					if(1 == EDGEPOS(gPanelObj.KeyMatric[S$KEYMATRIX_F8],KeyMatric[S$KEYMATRIX_F8]))
					{
					if(0 == bLevel3CalibHide)
					{
						if(ACTUATOR_ELECTRIC == gMachineFix.MoldR.Clamp.eActuatorType)
						{
							gPanelObj.SetPicture = PIC_CALIB_CLAMP_ENCODER;
						}
						else if(ACTUATOR_HYD == gMachineFix.MoldR.Clamp.eActuatorType )
						{
							gPanelObj.SetPicture = PIC_CALIB_CLAMP_LVDT;
						}
					}
				}
				if(1 == bLevel3CalibHide)gPanelObj.idxKeyPicture[S$KEYMATRIX_F8] = STATE_INACTIVE;

					//				gPanelObj.idxKeyPicture[S$KEYMATRIX_F7] = STATE_INACTIVE;
					//				gPanelObj.idxKeyPicture[S$KEYMATRIX_F8] = STATE_INACTIVE;
					gPanelObj.idxKeyPicture[S$KEYMATRIX_F9] = STATE_SUB_PAGE;
					if(1 == EDGEPOS(gPanelObj.KeyMatric[S$KEYMATRIX_F9],KeyMatric[S$KEYMATRIX_F9]))
					{
					if(gPanelObj.PasswordLevel > 3 && 1 == gTKcalib.Status)
					{
						gPanelObj.SetPicture = PIC_PROPORTION_VALVE;
					}
				}
				if(1 == bHidePropValvePage)gPanelObj.idxKeyPicture[S$KEYMATRIX_F9] = STATE_INACTIVE;

					gPanelObj.idxKeyPicture[S$KEYMATRIX_F10] = STATE_SUB_PAGE;
					if(1 == EDGEPOS(gPanelObj.KeyMatric[S$KEYMATRIX_F10],KeyMatric[S$KEYMATRIX_F10]))
					{
					gPanelObj.SetPicture = PIC_SCREEN_CALIBRATE;
				}

				gPanelObj.idxKeyPicture[S$KEYMATRIX_F11] = STATE_SUB_PAGE;
					if(1 == EDGEPOS(gPanelObj.KeyMatric[S$KEYMATRIX_F11],KeyMatric[S$KEYMATRIX_F11]))
					{
					if(gPanelObj.PasswordLevel > 2)gPanelObj.SetPicture = PIC_PV_LOG;
				}
				if(gPanelObj.PasswordLevel < 3)gPanelObj.idxKeyPicture[S$KEYMATRIX_F11] = STATE_INACTIVE;

					gPanelObj.idxKeyPicture[S$KEYMATRIX_F12] = STATE_SUB_PAGE;
					if(1 == EDGEPOS(gPanelObj.KeyMatric[S$KEYMATRIX_F12],KeyMatric[S$KEYMATRIX_F12]))
					{
					if(gPanelObj.PasswordLevel > 2)gPanelObj.SetPicture = PIC_LOG_INFO;
				}
				if(gPanelObj.PasswordLevel < 3)gPanelObj.idxKeyPicture[S$KEYMATRIX_F12] = STATE_INACTIVE;

					gPanelObj.idxKeyPicture[S$KEYMATRIX_F13] = STATE_SUB_PAGE;
					if(1 == EDGEPOS(gPanelObj.KeyMatric[S$KEYMATRIX_F13],KeyMatric[S$KEYMATRIX_F13]))
					{
					if(gPanelObj.PasswordLevel > 0)gPanelObj.SetPicture = PIC_INDUSTY_40;
				}
				if(gPanelObj.PasswordLevel < 1)gPanelObj.idxKeyPicture[S$KEYMATRIX_F13] = STATE_INACTIVE;

					gPanelObj.idxKeyPicture[S$KEYMATRIX_F14] = STATE_SUB_PAGE;
					if(1 == EDGEPOS(gPanelObj.KeyMatric[S$KEYMATRIX_F14],KeyMatric[S$KEYMATRIX_F14]))
					{
					if(gPanelObj.PasswordLevel > 0)gPanelObj.SetPicture = PIC_IP_CONFIG;
				}
				if(gPanelObj.PasswordLevel < 1)gPanelObj.idxKeyPicture[S$KEYMATRIX_F14] = STATE_INACTIVE;

					gPanelObj.idxKeyPicture[S$KEYMATRIX_F15] = STATE_SUB_PAGE;
					if(1 == EDGEPOS(gPanelObj.KeyMatric[S$KEYMATRIX_F15],KeyMatric[S$KEYMATRIX_F15]))
					{
					if(gPanelObj.PasswordLevel > 0)gPanelObj.SetPicture = PIC_VNC;
				}
				if(gPanelObj.PasswordLevel < 1)gPanelObj.idxKeyPicture[S$KEYMATRIX_F15] = STATE_INACTIVE;

					gPanelObj.idxKeyPicture[S$KEYMATRIX_F16] = STATE_SUB_PAGE;
					if(1 == EDGEPOS(gPanelObj.KeyMatric[S$KEYMATRIX_F16],KeyMatric[S$KEYMATRIX_F16]))
					{
					gPanelObj.SetPicture = PIC_PASSWORD_LOGIN;
				}

				if(1 == gPanelObj.KeyMatric[S$KEYMATRIX_TAB]&& 1 == gPanelObj.KeyMatric[S$KEYMATRIX_ENTER])
					{
					if(gPanelObj.PasswordLevel > 2)gPanelObj.SetPicture = PIC_DEFAULT_SET  ;
				}
				break;

			case PIC_SYSTEM_SET_1:
				if(ChangePageDly > 0)
				{
					ChangePageDly--;
					break;
				}

				gPanelObj.idxKeyPicture[S$KEYMATRIX_F1] = STATE_SUB_PAGE;
					if(1 == EDGEPOS(gPanelObj.KeyMatric[S$KEYMATRIX_F1],KeyMatric[S$KEYMATRIX_F1]))
					{
					gPanelObj.SetPicture = PIC_OVERVIEW;
				}

				gPanelObj.idxKeyPicture[S$KEYMATRIX_F2] = STATE_SUB_PAGE;
					if(1 == EDGEPOS(gPanelObj.KeyMatric[S$KEYMATRIX_F2],KeyMatric[S$KEYMATRIX_F2]))
					{
					gPanelObj.SetPicture = gPanelObj.OldPicture;
				}

				gPanelObj.idxKeyPicture[S$KEYMATRIX_F3] = STATE_ACTIVE;
					if(1 == EDGEPOS(gPanelObj.KeyMatric[S$KEYMATRIX_F3],KeyMatric[S$KEYMATRIX_F3]))
					{
					gPanelObj.SetPicture = PIC_SYSTEM_SET_2;
				}

				gPanelObj.idxKeyPicture[S$KEYMATRIX_F4] = STATE_SUB_PAGE;
					if(1 == EDGEPOS(gPanelObj.KeyMatric[S$KEYMATRIX_F4],KeyMatric[S$KEYMATRIX_F4]))
					{
					gPanelObj.SetPicture = PIC_ACCU_SETTING;
				}

				gPanelObj.idxKeyPicture[S$KEYMATRIX_F5] = STATE_SUB_PAGE;
					if(1 == EDGEPOS(gPanelObj.KeyMatric[S$KEYMATRIX_F5],KeyMatric[S$KEYMATRIX_F5]))
					{
					if(gPanelObj.PasswordLevel > 3)gPanelObj.SetPicture = PIC_OEM_SETTING_1;
				}
				if(gPanelObj.PasswordLevel <= 3)gPanelObj.idxKeyPicture[S$KEYMATRIX_F5] = STATE_INACTIVE;

					gPanelObj.idxKeyPicture[S$KEYMATRIX_F6] = STATE_SUB_PAGE;
					if(1 == EDGEPOS(gPanelObj.KeyMatric[S$KEYMATRIX_F6],KeyMatric[S$KEYMATRIX_F6]))
					{
					if(gPanelObj.PasswordLevel > 0)gPanelObj.SetPicture = PIC_PASSWORD_SET;
				}
				gPanelObj.idxKeyPicture[S$KEYMATRIX_F7] = STATE_SUB_PAGE;
					if(1 == EDGEPOS(gPanelObj.KeyMatric[S$KEYMATRIX_F7],KeyMatric[S$KEYMATRIX_F7]))
					{
					if(gPanelObj.PasswordLevel > 2)gPanelObj.SetPicture = PIC_PRESSURE_CALIBRATION ;
				}
				if(gPanelObj.PasswordLevel <= 2)gPanelObj.idxKeyPicture[S$KEYMATRIX_F7] = STATE_INACTIVE;
					//				gPanelObj.idxKeyPicture[S$KEYMATRIX_F7] = STATE_SUB_PAGE;
					//				if(1 == EDGEPOS(gPanelObj.KeyMatric[S$KEYMATRIX_F7],KeyMatric[S$KEYMATRIX_F7]))
					//				{
					//					if(0 == bLevel3CalibHide)
					//					{
					//						gPanelObj.SetPicture = PIC_MOLD_CALIBRATION;
					//					}
					//				}
					//				if(1 == bLevel3CalibHide)gPanelObj.idxKeyPicture[S$KEYMATRIX_F7] = STATE_INACTIVE;

					gPanelObj.idxKeyPicture[S$KEYMATRIX_F8] = STATE_SUB_PAGE;
					if(1 == EDGEPOS(gPanelObj.KeyMatric[S$KEYMATRIX_F8],KeyMatric[S$KEYMATRIX_F8]))
					{
					if(0 == bLevel3CalibHide)
					{
						if(ACTUATOR_ELECTRIC == gMachineFix.MoldR.Clamp.eActuatorType)
						{
							gPanelObj.SetPicture = PIC_CALIB_CLAMP_ENCODER;
						}
						else if(ACTUATOR_HYD == gMachineFix.MoldR.Clamp.eActuatorType )
						{
							gPanelObj.SetPicture = PIC_CALIB_CLAMP_LVDT;
						}
					}
				}
				if(1 == bLevel3CalibHide)gPanelObj.idxKeyPicture[S$KEYMATRIX_F8] = STATE_INACTIVE;

					//				gPanelObj.idxKeyPicture[S$KEYMATRIX_F7] = STATE_INACTIVE;
					//				gPanelObj.idxKeyPicture[S$KEYMATRIX_F8] = STATE_INACTIVE;

					gPanelObj.idxKeyPicture[S$KEYMATRIX_F9] = STATE_SUB_PAGE;
					if(1 == EDGEPOS(gPanelObj.KeyMatric[S$KEYMATRIX_F9],KeyMatric[S$KEYMATRIX_F9]))
					{
					if(gPanelObj.PasswordLevel > 3 && 1 == gTKcalib.Status)
					{
						gPanelObj.SetPicture = PIC_PROPORTION_VALVE;
					}
				}
				if(1 == bHidePropValvePage)gPanelObj.idxKeyPicture[S$KEYMATRIX_F9] = STATE_INACTIVE;

					gPanelObj.idxKeyPicture[S$KEYMATRIX_F10] = STATE_SUB_PAGE;
					if(1 == EDGEPOS(gPanelObj.KeyMatric[S$KEYMATRIX_F10],KeyMatric[S$KEYMATRIX_F10]))
					{
					gPanelObj.SetPicture = PIC_SCREEN_CALIBRATE;
				}

				gPanelObj.idxKeyPicture[S$KEYMATRIX_F11] = STATE_SUB_PAGE;
					if(1 == EDGEPOS(gPanelObj.KeyMatric[S$KEYMATRIX_F11],KeyMatric[S$KEYMATRIX_F11]))
					{
					if(gPanelObj.PasswordLevel > 2)gPanelObj.SetPicture = PIC_PV_LOG;
				}
				if(gPanelObj.PasswordLevel < 3)gPanelObj.idxKeyPicture[S$KEYMATRIX_F11] = STATE_INACTIVE;

					gPanelObj.idxKeyPicture[S$KEYMATRIX_F12] = STATE_SUB_PAGE;
					if(1 == EDGEPOS(gPanelObj.KeyMatric[S$KEYMATRIX_F12],KeyMatric[S$KEYMATRIX_F12]))
					{
					if(gPanelObj.PasswordLevel > 2)gPanelObj.SetPicture = PIC_LOG_INFO;
				}
				if(gPanelObj.PasswordLevel < 3)gPanelObj.idxKeyPicture[S$KEYMATRIX_F12] = STATE_INACTIVE;

					gPanelObj.idxKeyPicture[S$KEYMATRIX_F13] = STATE_SUB_PAGE;
					if(1 == EDGEPOS(gPanelObj.KeyMatric[S$KEYMATRIX_F13],KeyMatric[S$KEYMATRIX_F13]))
					{
					if(gPanelObj.PasswordLevel > 0)gPanelObj.SetPicture = PIC_INDUSTY_40;
				}
				if(gPanelObj.PasswordLevel < 1)gPanelObj.idxKeyPicture[S$KEYMATRIX_F13] = STATE_INACTIVE;

					gPanelObj.idxKeyPicture[S$KEYMATRIX_F14] = STATE_SUB_PAGE;
					if(1 == EDGEPOS(gPanelObj.KeyMatric[S$KEYMATRIX_F14],KeyMatric[S$KEYMATRIX_F14]))
					{
					if(gPanelObj.PasswordLevel > 0)gPanelObj.SetPicture = PIC_IP_CONFIG;
				}
				if(gPanelObj.PasswordLevel < 1)gPanelObj.idxKeyPicture[S$KEYMATRIX_F14] = STATE_INACTIVE;

					gPanelObj.idxKeyPicture[S$KEYMATRIX_F15] = STATE_SUB_PAGE;
					if(1 == EDGEPOS(gPanelObj.KeyMatric[S$KEYMATRIX_F15],KeyMatric[S$KEYMATRIX_F15]))
					{
					if(gPanelObj.PasswordLevel > 0)gPanelObj.SetPicture = PIC_VNC;
				}

				//						gPanelObj.idxKeyPicture[S$KEYMATRIX_F7] = STATE_INACTIVE;
				//            		gPanelObj.idxKeyPicture[S$KEYMATRIX_F8] = STATE_INACTIVE;
				//						gPanelObj.idxKeyPicture[S$KEYMATRIX_F8] = STATE_SUB_BUTTON;
				//						if(1 == EDGEPOS(gPanelObj.KeyMatric[S$KEYMATRIX_F8],KeyMatric[S$KEYMATRIX_F8]))
				//						{
				//						gMachineInfo.CycleTimes = 0;
				//						gCycleTimes             = 0;
				//						gMachineInfo.GoodBottles = 0;
				//					}

				//					gPanelObj.idxKeyPicture[S$KEYMATRIX_F9] = STATE_INACTIVE;
				//					gPanelObj.idxKeyPicture[S$KEYMATRIX_F10] = STATE_INACTIVE;
				//						gPanelObj.idxKeyPicture[S$KEYMATRIX_F10] = STATE_SUB_PAGE;
				//						if(1 == EDGEPOS(gPanelObj.KeyMatric[S$KEYMATRIX_F10],KeyMatric[S$KEYMATRIX_F10]))
				//						{
				//						gPanelObj.SetPicture = PIC_SCREEN_CALIBRATE;
				//					}
				//					gPanelObj.idxKeyPicture[S$KEYMATRIX_F11] = STATE_INACTIVE;
				//						gPanelObj.idxKeyPicture[S$KEYMATRIX_F12] = STATE_INACTIVE;
				//						gPanelObj.idxKeyPicture[S$KEYMATRIX_F13] = STATE_INACTIVE;
				//						gPanelObj.idxKeyPicture[S$KEYMATRIX_F14] = STATE_INACTIVE;
				//						gPanelObj.idxKeyPicture[S$KEYMATRIX_F15] = STATE_INACTIVE;

				gPanelObj.idxKeyPicture[S$KEYMATRIX_F16] = STATE_SUB_PAGE;
					if(1 == EDGEPOS(gPanelObj.KeyMatric[S$KEYMATRIX_F16],KeyMatric[S$KEYMATRIX_F16]))
					{
					gPanelObj.SetPicture = PIC_PASSWORD_LOGIN;
				}
				break;

			case PIC_SYSTEM_SET_2:
				if(ChangePageDly > 0)
				{
					ChangePageDly--;
					break;
				}

				gPanelObj.idxKeyPicture[S$KEYMATRIX_F1] = STATE_SUB_PAGE;
					if(1 == EDGEPOS(gPanelObj.KeyMatric[S$KEYMATRIX_F1],KeyMatric[S$KEYMATRIX_F1]))
					{
					gPanelObj.SetPicture = PIC_OVERVIEW;
				}

				gPanelObj.idxKeyPicture[S$KEYMATRIX_F2] = STATE_SUB_PAGE;
					if(1 == EDGEPOS(gPanelObj.KeyMatric[S$KEYMATRIX_F2],KeyMatric[S$KEYMATRIX_F2]))
					{
					gPanelObj.SetPicture = gPanelObj.OldPicture;
				}

				gPanelObj.idxKeyPicture[S$KEYMATRIX_F3] = STATE_SUB_PAGE;
					if(1 == EDGEPOS(gPanelObj.KeyMatric[S$KEYMATRIX_F3],KeyMatric[S$KEYMATRIX_F3]))
					{
					gPanelObj.SetPicture = PIC_SYSTEM_SET_1;
				}

				gPanelObj.idxKeyPicture[S$KEYMATRIX_F4] = STATE_ACTIVE;
					if(1 == EDGEPOS(gPanelObj.KeyMatric[S$KEYMATRIX_F4],KeyMatric[S$KEYMATRIX_F4]))
					{
					gPanelObj.SetPicture = PIC_ACCU_SETTING;
				}

				gPanelObj.idxKeyPicture[S$KEYMATRIX_F5] = STATE_SUB_PAGE;
					if(1 == EDGEPOS(gPanelObj.KeyMatric[S$KEYMATRIX_F5],KeyMatric[S$KEYMATRIX_F5]))
					{
					if(gPanelObj.PasswordLevel > 3)gPanelObj.SetPicture = PIC_OEM_SETTING_1;
				}
				if(gPanelObj.PasswordLevel <= 3)gPanelObj.idxKeyPicture[S$KEYMATRIX_F5] = STATE_INACTIVE;

					if(1 == EDGEPOS(gPanelObj.KeyMatric[S$KEYMATRIX_F6],KeyMatric[S$KEYMATRIX_F6]))
					{
					if(gPanelObj.PasswordLevel > 0)gPanelObj.SetPicture = PIC_PASSWORD_SET;
				}
				gPanelObj.idxKeyPicture[S$KEYMATRIX_F7] = STATE_SUB_PAGE;
					if(1 == EDGEPOS(gPanelObj.KeyMatric[S$KEYMATRIX_F7],KeyMatric[S$KEYMATRIX_F7]))
					{
					if(gPanelObj.PasswordLevel > 2)gPanelObj.SetPicture = PIC_PRESSURE_CALIBRATION ;
				}
				if(gPanelObj.PasswordLevel <= 2)gPanelObj.idxKeyPicture[S$KEYMATRIX_F7] = STATE_INACTIVE;
					//				gPanelObj.idxKeyPicture[S$KEYMATRIX_F7] = STATE_SUB_PAGE;
					//				if(1 == EDGEPOS(gPanelObj.KeyMatric[S$KEYMATRIX_F7],KeyMatric[S$KEYMATRIX_F7]))
					//				{
					//					if(0 == bLevel3CalibHide)
					//					{
					//						gPanelObj.SetPicture = PIC_MOLD_CALIBRATION;
					//					}
					//				}
					//				if(1 == bLevel3CalibHide)gPanelObj.idxKeyPicture[S$KEYMATRIX_F7] = STATE_INACTIVE;

					gPanelObj.idxKeyPicture[S$KEYMATRIX_F8] = STATE_SUB_PAGE;
					if(1 == EDGEPOS(gPanelObj.KeyMatric[S$KEYMATRIX_F8],KeyMatric[S$KEYMATRIX_F8]))
					{
					if(0 == bLevel3CalibHide)
					{
						if(ACTUATOR_ELECTRIC == gMachineFix.MoldR.Clamp.eActuatorType)
						{
							gPanelObj.SetPicture = PIC_CALIB_CLAMP_ENCODER;
						}
						else if(ACTUATOR_HYD == gMachineFix.MoldR.Clamp.eActuatorType )
						{
							gPanelObj.SetPicture = PIC_CALIB_CLAMP_LVDT;
						}
					}
				}
				if(1 == bLevel3CalibHide)gPanelObj.idxKeyPicture[S$KEYMATRIX_F8] = STATE_INACTIVE;

					//				gPanelObj.idxKeyPicture[S$KEYMATRIX_F7] = STATE_INACTIVE;
					//				gPanelObj.idxKeyPicture[S$KEYMATRIX_F8] = STATE_INACTIVE;

					gPanelObj.idxKeyPicture[S$KEYMATRIX_F9] = STATE_SUB_PAGE;
					if(1 == EDGEPOS(gPanelObj.KeyMatric[S$KEYMATRIX_F9],KeyMatric[S$KEYMATRIX_F9]))
					{
					if(gPanelObj.PasswordLevel > 3 && 1 == gTKcalib.Status)
					{
						gPanelObj.SetPicture = PIC_PROPORTION_VALVE;
					}
				}
				if(1 == bHidePropValvePage)gPanelObj.idxKeyPicture[S$KEYMATRIX_F9] = STATE_INACTIVE;

					gPanelObj.idxKeyPicture[S$KEYMATRIX_F10] = STATE_SUB_PAGE;
					if(1 == EDGEPOS(gPanelObj.KeyMatric[S$KEYMATRIX_F10],KeyMatric[S$KEYMATRIX_F10]))
					{
					gPanelObj.SetPicture = PIC_SCREEN_CALIBRATE;
				}

				gPanelObj.idxKeyPicture[S$KEYMATRIX_F11] = STATE_SUB_PAGE;
					if(1 == EDGEPOS(gPanelObj.KeyMatric[S$KEYMATRIX_F11],KeyMatric[S$KEYMATRIX_F11]))
					{
					if(gPanelObj.PasswordLevel > 2)gPanelObj.SetPicture = PIC_PV_LOG;
				}
				if(gPanelObj.PasswordLevel < 3)gPanelObj.idxKeyPicture[S$KEYMATRIX_F11] = STATE_INACTIVE;

					gPanelObj.idxKeyPicture[S$KEYMATRIX_F12] = STATE_SUB_PAGE;
					if(1 == EDGEPOS(gPanelObj.KeyMatric[S$KEYMATRIX_F12],KeyMatric[S$KEYMATRIX_F12]))
					{
					if(gPanelObj.PasswordLevel > 2)gPanelObj.SetPicture = PIC_LOG_INFO;
				}
				if(gPanelObj.PasswordLevel < 3)gPanelObj.idxKeyPicture[S$KEYMATRIX_F12] = STATE_INACTIVE;

					gPanelObj.idxKeyPicture[S$KEYMATRIX_F13] = STATE_SUB_PAGE;
					if(1 == EDGEPOS(gPanelObj.KeyMatric[S$KEYMATRIX_F13],KeyMatric[S$KEYMATRIX_F13]))
					{
					if(gPanelObj.PasswordLevel > 0)gPanelObj.SetPicture = PIC_INDUSTY_40;
				}
				if(gPanelObj.PasswordLevel < 1)gPanelObj.idxKeyPicture[S$KEYMATRIX_F13] = STATE_INACTIVE;

					gPanelObj.idxKeyPicture[S$KEYMATRIX_F14] = STATE_SUB_PAGE;
					if(1 == EDGEPOS(gPanelObj.KeyMatric[S$KEYMATRIX_F14],KeyMatric[S$KEYMATRIX_F14]))
					{
					if(gPanelObj.PasswordLevel > 0)gPanelObj.SetPicture = PIC_IP_CONFIG;
				}
				if(gPanelObj.PasswordLevel < 1)gPanelObj.idxKeyPicture[S$KEYMATRIX_F14] = STATE_INACTIVE;

					gPanelObj.idxKeyPicture[S$KEYMATRIX_F15] = STATE_SUB_PAGE;
					if(1 == EDGEPOS(gPanelObj.KeyMatric[S$KEYMATRIX_F15],KeyMatric[S$KEYMATRIX_F15]))
					{
					if(gPanelObj.PasswordLevel > 0)gPanelObj.SetPicture = PIC_VNC;
				}
				//						gPanelObj.idxKeyPicture[S$KEYMATRIX_F7] = STATE_SUB_BUTTON;
				//						if(1 == EDGEPOS(gPanelObj.KeyMatric[S$KEYMATRIX_F7],KeyMatric[S$KEYMATRIX_F7]))
				//						{
				//						gMachineFix.Option.AlarmTextMode  = !gMachineFix.Option.AlarmTextMode;
				//					}
				//
				//					gPanelObj.idxKeyPicture[S$KEYMATRIX_F8] = STATE_SUB_BUTTON;
				//						if(1 == EDGEPOS(gPanelObj.KeyMatric[S$KEYMATRIX_F8],KeyMatric[S$KEYMATRIX_F8]))
				//						{
				//						gMachineFix.Option.AlarmLedMode  = !gMachineFix.Option.AlarmLedMode;
				//					}
				//
				//					gPanelObj.idxKeyPicture[S$KEYMATRIX_F9] = STATE_SUB_BUTTON;
				//						if(1 == EDGEPOS(gPanelObj.KeyMatric[S$KEYMATRIX_F9],KeyMatric[S$KEYMATRIX_F9]))
				//						{
				//						/*gPwd.Language = ! gPwd.Language;*/
				//						gPanelObj.SetLanguage = gPanelObj.GetLanguage + 1;
				//						if(gPanelObj.SetLanguage > 2)gPanelObj.SetLanguage = 1;
				//					}
				//            		gPanelObj.idxKeyPicture[S$KEYMATRIX_F7] = STATE_INACTIVE;
				//					gPanelObj.idxKeyPicture[S$KEYMATRIX_F8] = STATE_INACTIVE;
				//					gPanelObj.idxKeyPicture[S$KEYMATRIX_F9] = STATE_INACTIVE;
				//					gPanelObj.idxKeyPicture[S$KEYMATRIX_F10] = STATE_INACTIVE;
				//						gPanelObj.idxKeyPicture[S$KEYMATRIX_F11] = STATE_INACTIVE;

				//						gPanelObj.idxKeyPicture[S$KEYMATRIX_F12] = STATE_SUB_BUTTON;
				//						if(1 == EDGEPOS(gPanelObj.KeyMatric[S$KEYMATRIX_F12],KeyMatric[S$KEYMATRIX_F12]))
				//						{
				//						if(1 == gRecipeOperate.usbDiskOk)gScreenShot.CmdScreenShotAll = 1;
				//					}
				//					gPanelObj.idxKeyPicture[S$KEYMATRIX_F12] = STATE_INACTIVE;
				//					gPanelObj.idxKeyPicture[S$KEYMATRIX_F13] = STATE_INACTIVE;
				//						gPanelObj.idxKeyPicture[S$KEYMATRIX_F14] = STATE_INACTIVE;
				//						gPanelObj.idxKeyPicture[S$KEYMATRIX_F15] = STATE_INACTIVE;

				gPanelObj.idxKeyPicture[S$KEYMATRIX_F16] = STATE_SUB_PAGE;
					if(1 == EDGEPOS(gPanelObj.KeyMatric[S$KEYMATRIX_F16],KeyMatric[S$KEYMATRIX_F16]))
					{
					gPanelObj.SetPicture = PIC_PASSWORD_LOGIN;
				}
				break;

			case PIC_SYSTEM_SET_3:
				if(ChangePageDly > 0)
				{
					ChangePageDly--;
					break;
				}

				gPanelObj.idxKeyPicture[S$KEYMATRIX_F1] = STATE_SUB_PAGE;
					if(1 == EDGEPOS(gPanelObj.KeyMatric[S$KEYMATRIX_F1],KeyMatric[S$KEYMATRIX_F1]))
					{
					gPanelObj.SetPicture = PIC_OVERVIEW;
				}

				gPanelObj.idxKeyPicture[S$KEYMATRIX_F2] = STATE_SUB_PAGE;
					if(1 == EDGEPOS(gPanelObj.KeyMatric[S$KEYMATRIX_F2],KeyMatric[S$KEYMATRIX_F2]))
					{
					gPanelObj.SetPicture = gPanelObj.OldPicture;
				}

				gPanelObj.idxKeyPicture[S$KEYMATRIX_F3] = STATE_SUB_PAGE;
					if(1 == EDGEPOS(gPanelObj.KeyMatric[S$KEYMATRIX_F3],KeyMatric[S$KEYMATRIX_F3]))
					{
					gPanelObj.SetPicture = PIC_SYSTEM_SET_1;
				}

				gPanelObj.idxKeyPicture[S$KEYMATRIX_F4] = STATE_ACTIVE;
					if(1 == EDGEPOS(gPanelObj.KeyMatric[S$KEYMATRIX_F4],KeyMatric[S$KEYMATRIX_F4]))
					{
					gPanelObj.SetPicture = PIC_SYSTEM_SET_2;
				}

				gPanelObj.idxKeyPicture[S$KEYMATRIX_F5] = STATE_SUB_PAGE;
					if(1 == EDGEPOS(gPanelObj.KeyMatric[S$KEYMATRIX_F5],KeyMatric[S$KEYMATRIX_F5]))
					{
					gPanelObj.SetPicture = PIC_OEM_SETTING_1;
				}

				if(1 == EDGEPOS(gPanelObj.KeyMatric[S$KEYMATRIX_F6],KeyMatric[S$KEYMATRIX_F6]))
					{
					if(gPanelObj.PasswordLevel > 0)gPanelObj.SetPicture = PIC_PASSWORD_SET;
				}
				gPanelObj.idxKeyPicture[S$KEYMATRIX_F7] = STATE_SUB_PAGE;
					if(1 == EDGEPOS(gPanelObj.KeyMatric[S$KEYMATRIX_F7],KeyMatric[S$KEYMATRIX_F7]))
					{
					if(gPanelObj.PasswordLevel > 2)gPanelObj.SetPicture = PIC_PRESSURE_CALIBRATION ;
				}
				if(gPanelObj.PasswordLevel <= 2)gPanelObj.idxKeyPicture[S$KEYMATRIX_F7] = STATE_INACTIVE;
					//				gPanelObj.idxKeyPicture[S$KEYMATRIX_F7] = STATE_SUB_PAGE;
					//				if(1 == EDGEPOS(gPanelObj.KeyMatric[S$KEYMATRIX_F7],KeyMatric[S$KEYMATRIX_F7]))
					//				{
					//					if(0 == bLevel3CalibHide)
					//					{
					//						gPanelObj.SetPicture = PIC_MOLD_CALIBRATION;
					//					}
					//				}
					//				if(1 == bLevel3CalibHide)gPanelObj.idxKeyPicture[S$KEYMATRIX_F7] = STATE_INACTIVE;

					gPanelObj.idxKeyPicture[S$KEYMATRIX_F8] = STATE_SUB_PAGE;
					if(1 == EDGEPOS(gPanelObj.KeyMatric[S$KEYMATRIX_F8],KeyMatric[S$KEYMATRIX_F8]))
					{
					if(0 == bLevel3CalibHide)
					{
						if(ACTUATOR_ELECTRIC == gMachineFix.MoldR.Clamp.eActuatorType)
						{
							gPanelObj.SetPicture = PIC_CALIB_CLAMP_ENCODER;
						}
						else if(ACTUATOR_HYD == gMachineFix.MoldR.Clamp.eActuatorType )
						{
							gPanelObj.SetPicture = PIC_CALIB_CLAMP_LVDT;
						}
					}
				}
				if(1 == bLevel3CalibHide)gPanelObj.idxKeyPicture[S$KEYMATRIX_F8] = STATE_INACTIVE;

					//				gPanelObj.idxKeyPicture[S$KEYMATRIX_F7] = STATE_INACTIVE;
					//				gPanelObj.idxKeyPicture[S$KEYMATRIX_F8] = STATE_INACTIVE;
					gPanelObj.idxKeyPicture[S$KEYMATRIX_F9] = STATE_SUB_PAGE;

					if(1 == EDGEPOS(gPanelObj.KeyMatric[S$KEYMATRIX_F9],KeyMatric[S$KEYMATRIX_F9]))
					{
					if(gPanelObj.PasswordLevel > 3 && 1 == gTKcalib.Status)
					{
						gPanelObj.SetPicture = PIC_PROPORTION_VALVE;
					}
				}
				if(1 == bHidePropValvePage)gPanelObj.idxKeyPicture[S$KEYMATRIX_F9] = STATE_INACTIVE;

					gPanelObj.idxKeyPicture[S$KEYMATRIX_F10] = STATE_SUB_PAGE;
					if(1 == EDGEPOS(gPanelObj.KeyMatric[S$KEYMATRIX_F10],KeyMatric[S$KEYMATRIX_F10]))
					{
					gPanelObj.SetPicture = PIC_SCREEN_CALIBRATE;
				}

				gPanelObj.idxKeyPicture[S$KEYMATRIX_F11] = STATE_SUB_PAGE;
					if(1 == EDGEPOS(gPanelObj.KeyMatric[S$KEYMATRIX_F11],KeyMatric[S$KEYMATRIX_F11]))
					{
					if(gPanelObj.PasswordLevel > 2)gPanelObj.SetPicture = PIC_PV_LOG;
				}
				if(gPanelObj.PasswordLevel < 3)gPanelObj.idxKeyPicture[S$KEYMATRIX_F11] = STATE_INACTIVE;

					gPanelObj.idxKeyPicture[S$KEYMATRIX_F12] = STATE_SUB_PAGE;
					if(1 == EDGEPOS(gPanelObj.KeyMatric[S$KEYMATRIX_F12],KeyMatric[S$KEYMATRIX_F12]))
					{
					if(gPanelObj.PasswordLevel > 2)gPanelObj.SetPicture = PIC_LOG_INFO;
				}
				if(gPanelObj.PasswordLevel < 3)gPanelObj.idxKeyPicture[S$KEYMATRIX_F12] = STATE_INACTIVE;

					gPanelObj.idxKeyPicture[S$KEYMATRIX_F13] = STATE_SUB_PAGE;
					if(1 == EDGEPOS(gPanelObj.KeyMatric[S$KEYMATRIX_F13],KeyMatric[S$KEYMATRIX_F13]))
					{
					if(gPanelObj.PasswordLevel > 0)gPanelObj.SetPicture = PIC_INDUSTY_40;
				}
				if(gPanelObj.PasswordLevel < 1)gPanelObj.idxKeyPicture[S$KEYMATRIX_F13] = STATE_INACTIVE;

					gPanelObj.idxKeyPicture[S$KEYMATRIX_F14] = STATE_SUB_PAGE;
					if(1 == EDGEPOS(gPanelObj.KeyMatric[S$KEYMATRIX_F14],KeyMatric[S$KEYMATRIX_F14]))
					{
					if(gPanelObj.PasswordLevel > 0)gPanelObj.SetPicture = PIC_IP_CONFIG;
				}
				if(gPanelObj.PasswordLevel < 1)gPanelObj.idxKeyPicture[S$KEYMATRIX_F14] = STATE_INACTIVE;

					gPanelObj.idxKeyPicture[S$KEYMATRIX_F15] = STATE_SUB_PAGE;
					if(1 == EDGEPOS(gPanelObj.KeyMatric[S$KEYMATRIX_F15],KeyMatric[S$KEYMATRIX_F15]))
					{
					if(gPanelObj.PasswordLevel > 0)gPanelObj.SetPicture = PIC_VNC;
				}
				//						gPanelObj.idxKeyPicture[S$KEYMATRIX_F7] = STATE_SUB_BUTTON;
				//						if(1 == EDGEPOS(gPanelObj.KeyMatric[S$KEYMATRIX_F7],KeyMatric[S$KEYMATRIX_F7]))
				//						{
				//						gMachineFix.Option.AlarmTextMode  = !gMachineFix.Option.AlarmTextMode;
				//					}
				//
				//					gPanelObj.idxKeyPicture[S$KEYMATRIX_F8] = STATE_SUB_BUTTON;
				//						if(1 == EDGEPOS(gPanelObj.KeyMatric[S$KEYMATRIX_F8],KeyMatric[S$KEYMATRIX_F8]))
				//						{
				//						gMachineFix.Option.AlarmLedMode  = !gMachineFix.Option.AlarmLedMode;
				//					}
				//
				//					gPanelObj.idxKeyPicture[S$KEYMATRIX_F9] = STATE_SUB_BUTTON;
				//						if(1 == EDGEPOS(gPanelObj.KeyMatric[S$KEYMATRIX_F9],KeyMatric[S$KEYMATRIX_F9]))
				//						{
				//						/*gPwd.Language = ! gPwd.Language;*/
				//						gPanelObj.SetLanguage = gPanelObj.GetLanguage + 1;
				//						if(gPanelObj.SetLanguage > 2)gPanelObj.SetLanguage = 1;
				//					}
				//            		gPanelObj.idxKeyPicture[S$KEYMATRIX_F7] = STATE_INACTIVE;
				//					gPanelObj.idxKeyPicture[S$KEYMATRIX_F8] = STATE_INACTIVE;
				//					gPanelObj.idxKeyPicture[S$KEYMATRIX_F9] = STATE_INACTIVE;
				//					gPanelObj.idxKeyPicture[S$KEYMATRIX_F10] = STATE_INACTIVE;
				//						gPanelObj.idxKeyPicture[S$KEYMATRIX_F11] = STATE_INACTIVE;

				//						gPanelObj.idxKeyPicture[S$KEYMATRIX_F12] = STATE_SUB_BUTTON;
				//						if(1 == EDGEPOS(gPanelObj.KeyMatric[S$KEYMATRIX_F12],KeyMatric[S$KEYMATRIX_F12]))
				//						{
				//						if(1 == gRecipeOperate.usbDiskOk)gScreenShot.CmdScreenShotAll = 1;
				//					}
				//					gPanelObj.idxKeyPicture[S$KEYMATRIX_F12] = STATE_INACTIVE;
				//					gPanelObj.idxKeyPicture[S$KEYMATRIX_F13] = STATE_INACTIVE;
				//						gPanelObj.idxKeyPicture[S$KEYMATRIX_F14] = STATE_INACTIVE;
				//						gPanelObj.idxKeyPicture[S$KEYMATRIX_F15] = STATE_INACTIVE;

				gPanelObj.idxKeyPicture[S$KEYMATRIX_F16] = STATE_SUB_PAGE;
					if(1 == EDGEPOS(gPanelObj.KeyMatric[S$KEYMATRIX_F16],KeyMatric[S$KEYMATRIX_F16]))
					{
					gPanelObj.SetPicture = PIC_PASSWORD_LOGIN;
				}
				break;

			case PIC_OEM_SETTING_1:  // 180
			case PIC_OEM_SETTING_2:  // 181
			case PIC_OEM_SETTING_3:  // 182
			case PIC_OEM_SETTING_4:  // 183
			case PIC_OEM_SETTING_10:  // 189

				if(ChangePageDly > 0)
				{
					ChangePageDly--;
					break;
				}

				gPanelObj.idxKeyPicture[S$KEYMATRIX_F1] = STATE_SUB_PAGE;
					if(1 == EDGEPOS(gPanelObj.KeyMatric[S$KEYMATRIX_F1],KeyMatric[S$KEYMATRIX_F1]))
					{
					gPanelObj.SetPicture = PIC_OVERVIEW;
				}

				gPanelObj.idxKeyPicture[S$KEYMATRIX_F2] = STATE_SUB_PAGE;
					if(1 == EDGEPOS(gPanelObj.KeyMatric[S$KEYMATRIX_F2],KeyMatric[S$KEYMATRIX_F2]))
					{
					gPanelObj.SetPicture = gPanelObj.OldPicture;
				}

				gPanelObj.idxKeyPicture[S$KEYMATRIX_F3] = STATE_SUB_PAGE;
					if(1 == EDGEPOS(gPanelObj.KeyMatric[S$KEYMATRIX_F3],KeyMatric[S$KEYMATRIX_F3]))
					{
					gPanelObj.SetPicture = PIC_OEM_SETTING_1;
				}

				gPanelObj.idxKeyPicture[S$KEYMATRIX_F4] = STATE_SUB_PAGE;
					if(1 == EDGEPOS(gPanelObj.KeyMatric[S$KEYMATRIX_F4],KeyMatric[S$KEYMATRIX_F4]))
					{
					gPanelObj.SetPicture = PIC_OEM_SETTING_2;
				}

				gPanelObj.idxKeyPicture[S$KEYMATRIX_F5] = STATE_SUB_PAGE;
					if(1 == EDGEPOS(gPanelObj.KeyMatric[S$KEYMATRIX_F5],KeyMatric[S$KEYMATRIX_F5]))
					{
					gPanelObj.SetPicture = PIC_OEM_SETTING_3;
				}

				gPanelObj.idxKeyPicture[S$KEYMATRIX_F6] = STATE_SUB_PAGE;
					if(1 == EDGEPOS(gPanelObj.KeyMatric[S$KEYMATRIX_F6],KeyMatric[S$KEYMATRIX_F6]))
					{
					gPanelObj.SetPicture = PIC_OEM_SETTING_4;
				}
				gPanelObj.idxKeyPicture[S$KEYMATRIX_F7] = STATE_INACTIVE;
					gPanelObj.idxKeyPicture[S$KEYMATRIX_F8] = STATE_INACTIVE;
					gPanelObj.idxKeyPicture[S$KEYMATRIX_F9] = STATE_INACTIVE;
					gPanelObj.idxKeyPicture[S$KEYMATRIX_F10] = STATE_INACTIVE;
					gPanelObj.idxKeyPicture[S$KEYMATRIX_F11] = STATE_INACTIVE;

					gPanelObj.idxKeyPicture[S$KEYMATRIX_F12] = STATE_SUB_PAGE;
					if(1 == EDGEPOS(gPanelObj.KeyMatric[S$KEYMATRIX_F12],KeyMatric[S$KEYMATRIX_F12]))
					{
					gPanelObj.SetPicture = PIC_OEM_SETTING_10;
				}
				gPanelObj.idxKeyPicture[S$KEYMATRIX_F13] = STATE_INACTIVE;
					gPanelObj.idxKeyPicture[S$KEYMATRIX_F14] = STATE_INACTIVE;
					gPanelObj.idxKeyPicture[S$KEYMATRIX_F15] = STATE_INACTIVE;

					gPanelObj.idxKeyPicture[S$KEYMATRIX_F16] = STATE_SUB_PAGE;
					if(1 == EDGEPOS(gPanelObj.KeyMatric[S$KEYMATRIX_F16],KeyMatric[S$KEYMATRIX_F16]))
					{
					gPanelObj.SetPicture = PIC_PASSWORD_LOGIN;
				}
				break;

			case PIC_IP_CONFIG: //135
			case PIC_PRESSURE_CALIBRATION:  //134
			case PIC_LOG_INFO:  //137
			case PIC_INDUSTY_40:	//125
			case PIC_VNC:	//138
			case PIC_PROPORTION_VALVE: //133
			case PIC_ACCU_SETTING: //68
				if(ChangePageDly > 0)
				{
					ChangePageDly--;
					break;
				}

				gPanelObj.idxKeyPicture[S$KEYMATRIX_F1] = STATE_SUB_PAGE;
					if(1 == EDGEPOS(gPanelObj.KeyMatric[S$KEYMATRIX_F1],KeyMatric[S$KEYMATRIX_F1]))
					{
					gPanelObj.SetPicture = PIC_OVERVIEW;
				}

				gPanelObj.idxKeyPicture[S$KEYMATRIX_F2] = STATE_SUB_PAGE;
					if(1 == EDGEPOS(gPanelObj.KeyMatric[S$KEYMATRIX_F2],KeyMatric[S$KEYMATRIX_F2]))
					{
					gPanelObj.SetPicture = gPanelObj.OldPicture;
				}

				gPanelObj.idxKeyPicture[S$KEYMATRIX_F3] = STATE_SUB_PAGE;
					if(1 == EDGEPOS(gPanelObj.KeyMatric[S$KEYMATRIX_F3],KeyMatric[S$KEYMATRIX_F3]))
					{
					gPanelObj.SetPicture = PIC_SYSTEM_SET_1;
				}

				gPanelObj.idxKeyPicture[S$KEYMATRIX_F4] = STATE_SUB_PAGE;
					if(1 == EDGEPOS(gPanelObj.KeyMatric[S$KEYMATRIX_F4],KeyMatric[S$KEYMATRIX_F4]))
					{
					gPanelObj.SetPicture = PIC_ACCU_SETTING;
				}
```
